LIN {X 0,Y 411.995,Z 195.318,A -85,B 0,C 180,E1 -10499.219,E2 -10499.219} C_VEL
LIN {X 0,Y 411.545,Z 202.189,A -85,B 0,C 180,E1 -10502.624,E2 -10502.624} C_VEL
LIN {X 0,Y 411.166,Z 208.718,A -85,B 0,C 180,E1 -10505.781,E2 -10505.781} C_VEL
LIN {X 0,Y 410.854,Z 215.36,A -85,B 0,C 180,E1 -10508.947,E2 -10508.947} C_VEL
LIN {X 0,Y 410.565,Z 222.705,A -85,B 0,C 180,E1 -10512.421,E2 -10512.421} C_VEL
LIN {X 0,Y 412.997,Z 235.986,A -85,B 0,C 180,E1 -10512.93,E2 -10512.93} C_VEL
LIN {X 0,Y 414.87,Z 248.726,A -85,B 0,C 180,E1 -10513.605,E2 -10513.605} C_VEL
LIN {X 0,Y 414.456,Z 259.342,A -85,B 0,C 180,E1 -10514.257,E2 -10514.257} C_VEL
LIN {X 0,Y 413.6,Z 271.793,A -85,B 0,C 180,E1 -10515.233,E2 -10515.233} C_VEL
LIN {X 0,Y 412.816,Z 282.706,A -85,B 0,C 180,E1 -10516.337,E2 -10516.337} C_VEL
LIN {X 0,Y 412.22,Z 291.609,A -85,B 0,C 180,E1 -10517.445,E2 -10517.445} C_VEL
LIN {X 0,Y 411.418,Z 301.28,A -85,B 0,C 180,E1 -10518.92,E2 -10518.92} C_VEL
LIN {X 0,Y 410.866,Z 308.982,A -85,B 0,C 180,E1 -10520.399,E2 -10520.399} C_VEL
LIN {X 0,Y 410.366,Z 316.083,A -85,B 0,C 180,E1 -10522.125,E2 -10522.125} C_VEL
LIN {X 0,Y 410.126,Z 320.996,A -85,B 0,C 180,E1 -10523.669,E2 -10523.669} C_VEL
LIN {X 0,Y 410.061,Z 324.424,A -85,B 0,C 180,E1 -10525.084,E2 -10525.084} C_VEL
LIN {X 0,Y 409.943,Z 326.285,A -85,B 0,C 180,E1 -10526.068,E2 -10526.068} C_VEL
LIN {X 0,Y 409.963,Z 328.683,A -85,B 0,C 180,E1 -10528.035,E2 -10528.035} C_VEL
LIN {X 0,Y 409.919,Z 329.291,A -85,B 0,C 180,E1 -10529.017,E2 -10529.017} C_VEL
LIN {X 0,Y 409.888,Z 329.507,A -85,B 0,C 180,E1 -10530,E2 -10530} C_VEL
LIN {X 0,Y 409.918,Z 329.292,A -85,B 0,C 180,E1 -10530.982,E2 -10530.982} C_VEL
LIN {X 0,Y 409.963,Z 328.685,A -85,B 0,C 180,E1 -10531.965,E2 -10531.965} C_VEL
LIN {X 0,Y 409.943,Z 326.29,A -85,B 0,C 180,E1 -10533.932,E2 -10533.932} C_VEL
LIN {X 0,Y 410.063,Z 323.353,A -85,B 0,C 180,E1 -10535.409,E2 -10535.409} C_VEL
LIN {X 0,Y 410.198,Z 319.375,A -85,B 0,C 180,E1 -10536.888,E2 -10536.888} C_VEL
LIN {X 0,Y 410.575,Z 313.264,A -85,B 0,C 180,E1 -10538.614,E2 -10538.614} C_VEL
LIN {X 0,Y 411.025,Z 306.584,A -85,B 0,C 180,E1 -10540.094,E2 -10540.094} C_VEL
LIN {X 0,Y 411.628,Z 298.299,A -85,B 0,C 180,E1 -10541.573,E2 -10541.573} C_VEL
LIN {X 0,Y 412.349,Z 289.811,A -85,B 0,C 180,E1 -10542.801,E2 -10542.801} C_VEL
LIN {X 0,Y 413.082,Z 279.223,A -85,B 0,C 180,E1 -10544.041,E2 -10544.041} C_VEL
LIN {X 0,Y 413.869,Z 267.514,A -85,B 0,C 180,E1 -10545.134,E2 -10545.134} C_VEL
LIN {X 0,Y 414.693,Z 255.785,A -85,B 0,C 180,E1 -10545.977,E2 -10545.977} C_VEL
LIN {X 0,Y 414.853,Z 248.666,A -85,B 0,C 180,E1 -10546.398,E2 -10546.398} C_VEL
LIN {X 0,Y 412.873,Z 235.293,A -85,B 0,C 180,E1 -10547.101,E2 -10547.101} C_VEL
LIN {X 0,Y 410.566,Z 222.705,A -85,B 0,C 180,E1 -10547.578,E2 -10547.578} C_VEL
LIN {X 0,Y 410.856,Z 215.362,A -85,B 0,C 180,E1 -10551.052,E2 -10551.052} C_VEL
LIN {X 0,Y 411.17,Z 208.721,A -85,B 0,C 180,E1 -10554.219,E2 -10554.219} C_VEL
LIN {X 0,Y 411.553,Z 202.008,A -85,B 0,C 180,E1 -10557.456,E2 -10557.456} C_VEL
LIN {X 0,Y 412.003,Z 195.293,A -85,B 0,C 180,E1 -10560.78,E2 -10560.78} C_VEL
LIN {X 0,Y 412.452,Z 188.615,A -85,B 0,C 180,E1 -10564.215,E2 -10564.215} C_VEL
LIN {X 0,Y 412.517,Z 185.292,A -85,B 0,C 180,E1 -10565.999,E2 -10565.999} C_VEL
LIN {X 0,Y 412.084,Z 181.164,A -85,B 0,C 180,E1 -10568.324,E2 -10568.324} C_VEL
LIN {X 0,Y 411.209,Z 176.266,A -85,B 0,C 180,E1 -10571.316,E2 -10571.316} C_VEL
LIN {X 0,Y 411.175,Z 176.269,A -85,B 0,C 180,E1 -10574.49,E2 -10574.49} C_VEL
LIN {X 0,Y 411.175,Z 176.267,A -85,B 0,C 180,E1 -10578.194,E2 -10578.194} C_VEL
LIN {X 0,Y 411.201,Z 176.264,A -85,B 0,C 180,E1 -10580.774,E2 -10580.774} C_VEL
LIN {X 0,Y 411.193,Z 176.267,A -85,B 0,C 180,E1 -10584.471,E2 -10584.471} C_VEL
LIN {X 0,Y 411.205,Z 176.263,A -85,B 0,C 180,E1 -10586.873,E2 -10586.873} C_VEL
LIN {X 0,Y 411.231,Z 176.26,A -85,B 0,C 180,E1 -10590.644,E2 -10590.644} C_VEL
LIN {X 0,Y 411.235,Z 176.26,A -85,B 0,C 180,E1 -10593.619,E2 -10593.619} C_VEL
LIN {X 0,Y 411.193,Z 176.262,A -85,B 0,C 180,E1 -10596.852,E2 -10596.852} C_VEL
LIN {X 0,Y 411.213,Z 176.263,A -85,B 0,C 180,E1 -10600.05,E2 -10600.05} C_VEL
LIN {X 0,Y 411.261,Z 176.257,A -85,B 0,C 180,E1 -10603.131,E2 -10603.131} C_VEL
LIN {X 0,Y 411.303,Z 176.251,A -85,B 0,C 180,E1 -10606.896,E2 -10606.896} C_VEL
LIN {X 0,Y 411.285,Z 176.251,A -85,B 0,C 180,E1 -10610.161,E2 -10610.161} C_VEL
LIN {X 0,Y 411.389,Z 176.244,A -85,B 0,C 180,E1 -10613.132,E2 -10613.132} C_VEL
LIN {X 0,Y 411.298,Z 176.254,A -85,B 0,C 180,E1 -10615.099,E2 -10615.099} C_VEL
LIN {X 0,Y 411.509,Z 176.224,A -85,B 0,C 180,E1 -10618.043,E2 -10618.043} C_VEL
LIN {X 0,Y 411.64,Z 176.208,A -85,B 0,C 180,E1 -10620,E2 -10620} C_VEL
LIN {X 0,Y 411.453,Z 176.235,A -85,B 0,C 180,E1 -10622.937,E2 -10622.937} C_VEL
LIN {X 0,Y 411.388,Z 176.239,A -85,B 0,C 180,E1 -10626.574,E2 -10626.574} C_VEL
LIN {X 0,Y 411.286,Z 176.251,A -85,B 0,C 180,E1 -10629.839,E2 -10629.839} C_VEL
LIN {X 0,Y 411.303,Z 176.249,A -85,B 0,C 180,E1 -10633.104,E2 -10633.104} C_VEL
LIN {X 0,Y 411.255,Z 176.256,A -85,B 0,C 180,E1 -10636.889,E2 -10636.889} C_VEL
LIN {X 0,Y 411.229,Z 176.263,A -85,B 0,C 180,E1 -10639.987,E2 -10639.987} C_VEL
LIN {X 0,Y 411.2,Z 176.262,A -85,B 0,C 180,E1 -10643.148,E2 -10643.148} C_VEL
LIN {X 0,Y 411.235,Z 176.258,A -85,B 0,C 180,E1 -10646.381,E2 -10646.381} C_VEL
LIN {X 0,Y 411.199,Z 176.266,A -85,B 0,C 180,E1 -10649.713,E2 -10649.713} C_VEL
LIN {X 0,Y 411.205,Z 176.265,A -85,B 0,C 180,E1 -10653.156,E2 -10653.156} C_VEL
LIN {X 0,Y 411.187,Z 176.264,A -85,B 0,C 180,E1 -10656.552,E2 -10656.552} C_VEL
LIN {X 0,Y 411.198,Z 176.263,A -85,B 0,C 180,E1 -10659.726,E2 -10659.726} C_VEL
LIN {X 0,Y 411.172,Z 176.269,A -85,B 0,C 180,E1 -10663.134,E2 -10663.134} C_VEL
LIN {X 0,Y 411.168,Z 176.266,A -85,B 0,C 180,E1 -10665.881,E2 -10665.881} C_VEL
LIN {X 0,Y 411.163,Z 176.271,A -85,B 0,C 180,E1 -10668.772,E2 -10668.772} C_VEL
LIN {X 0,Y 411.185,Z 176.265,A -85,B 0,C 180,E1 -10672.026,E2 -10672.026} C_VEL
LIN {X 0,Y 411.148,Z 176.274,A -85,B 0,C 180,E1 -10673.456,E2 -10673.456} C_VEL
LIN {X 0,Y 411.077,Z 176.794,A -85,B 0,C 180,E1 -10674.46,E2 -10674.46} C_VEL
LIN {X 0,Y 411.058,Z 179.773,A -85,B 0,C 180,E1 -10676.906,E2 -10676.906} C_VEL
LIN {X 0,Y 410.962,Z 182.568,A -85,B 0,C 180,E1 -10679.134,E2 -10679.134} C_VEL
LIN {X 0,Y 410.777,Z 186.857,A -85,B 0,C 180,E1 -10682.488,E2 -10682.488} C_VEL
LIN {X 0,Y 410.625,Z 191.146,A -85,B 0,C 180,E1 -10685.747,E2 -10685.747} C_VEL
LIN {X 0,Y 410.456,Z 195.501,A -85,B 0,C 180,E1 -10688.927,E2 -10688.927} C_VEL
LIN {X 0,Y 410.314,Z 199.943,A -85,B 0,C 180,E1 -10692.043,E2 -10692.043} C_VEL
LIN {X 0,Y 410.322,Z 200.711,A -85,B 0,C 180,E1 -10692.492,E2 -10692.492} C_VEL
LIN {X 0,Y 413.415,Z 213.717,A -85,B 0,C 180,E1 -10693.057,E2 -10693.057} C_VEL
LIN {X 0,Y 415.382,Z 224.05,A -85,B 0,C 180,E1 -10693.632,E2 -10693.632} C_VEL
LIN {X 0,Y 414.694,Z 236.478,A -85,B 0,C 180,E1 -10694.393,E2 -10694.393} C_VEL
LIN {X 0,Y 414.053,Z 247.239,A -85,B 0,C 180,E1 -10695.25,E2 -10695.25} C_VEL
LIN {X 0,Y 413.373,Z 258.203,A -85,B 0,C 180,E1 -10696.356,E2 -10696.356} C_VEL
LIN {X 0,Y 412.634,Z 267.106,A -85,B 0,C 180,E1 -10697.458,E2 -10697.458} C_VEL
LIN {X 0,Y 412.026,Z 275.27,A -85,B 0,C 180,E1 -10698.688,E2 -10698.688} C_VEL
LIN {X 0,Y 411.384,Z 283.268,A -85,B 0,C 180,E1 -10700.164,E2 -10700.164} C_VEL
LIN {X 0,Y 410.825,Z 289.69,A -85,B 0,C 180,E1 -10701.639,E2 -10701.639} C_VEL
LIN {X 0,Y 410.499,Z 295.069,A -85,B 0,C 180,E1 -10703.217,E2 -10703.217} C_VEL
LIN {X 0,Y 410.287,Z 298.734,A -85,B 0,C 180,E1 -10704.594,E2 -10704.594} C_VEL
LIN {X 0,Y 410.085,Z 301.656,A -85,B 0,C 180,E1 -10706.069,E2 -10706.069} C_VEL
LIN {X 0,Y 410.088,Z 303.054,A -85,B 0,C 180,E1 -10707.053,E2 -10707.053} C_VEL
LIN {X 0,Y 409.94,Z 304.665,A -85,B 0,C 180,E1 -10709.018,E2 -10709.018} C_VEL
LIN {X 0,Y 409.928,Z 304.899,A -85,B 0,C 180,E1 -10710,E2 -10710} C_VEL
LIN {X 0,Y 409.94,Z 304.711,A -85,B 0,C 180,E1 -10710.983,E2 -10710.983} C_VEL
LIN {X 0,Y 410.088,Z 303.159,A -85,B 0,C 180,E1 -10712.947,E2 -10712.947} C_VEL
LIN {X 0,Y 410.081,Z 301.806,A -85,B 0,C 180,E1 -10713.931,E2 -10713.931} C_VEL
LIN {X 0,Y 410.281,Z 298.941,A -85,B 0,C 180,E1 -10715.406,E2 -10715.406} C_VEL
LIN {X 0,Y 410.502,Z 295.058,A -85,B 0,C 180,E1 -10716.883,E2 -10716.883} C_VEL
LIN {X 0,Y 410.803,Z 290.048,A -85,B 0,C 180,E1 -10718.362,E2 -10718.362} C_VEL
LIN {X 0,Y 411,Z 287.371,A -85,B 0,C 180,E1 -10719.027,E2 -10719.027} C_VEL
LIN {X 0,Y 410.607,Z 284.395,A -85,B 0,C 180,E1 -10719.738,E2 -10719.738} C_VEL
LIN {X 0,Y 408.245,Z 279.193,A -85,B 0,C 180,E1 -10720.875,E2 -10720.875} C_VEL
LIN {X 0,Y 405.913,Z 273.342,A -85,B 0,C 180,E1 -10721.956,E2 -10721.956} C_VEL
LIN {X 0,Y 405.565,Z 269.345,A -85,B 0,C 180,E1 -10722.571,E2 -10722.571} C_VEL
LIN {X 0,Y 406.415,Z 259.228,A -85,B 0,C 180,E1 -10723.883,E2 -10723.883} C_VEL
LIN {X 0,Y 407.141,Z 248.492,A -85,B 0,C 180,E1 -10725.007,E2 -10725.007} C_VEL
LIN {X 0,Y 407.865,Z 238.022,A -85,B 0,C 180,E1 -10725.876,E2 -10725.876} C_VEL
LIN {X 0,Y 408.549,Z 225.844,A -85,B 0,C 180,E1 -10726.658,E2 -10726.658} C_VEL
LIN {X 0,Y 406.426,Z 214.142,A -85,B 0,C 180,E1 -10727.333,E2 -10727.333} C_VEL
LIN {X 0,Y 403.243,Z 200.765,A -85,B 0,C 180,E1 -10727.947,E2 -10727.947} C_VEL
LIN {X 0,Y 403.339,Z 197.299,A -85,B 0,C 180,E1 -10730.395,E2 -10730.395} C_VEL
LIN {X 0,Y 403.506,Z 192.933,A -85,B 0,C 180,E1 -10733.616,E2 -10733.616} C_VEL
LIN {X 0,Y 403.701,Z 188.588,A -85,B 0,C 180,E1 -10736.913,E2 -10736.913} C_VEL
LIN {X 0,Y 403.872,Z 184.3,A -85,B 0,C 180,E1 -10740.308,E2 -10740.308} C_VEL
LIN {X 0,Y 404.054,Z 179.961,A -85,B 0,C 180,E1 -10743.821,E2 -10743.821} C_VEL
LIN {X 0,Y 404.059,Z 177.157,A -85,B 0,C 180,E1 -10746.255,E2 -10746.255} C_VEL
LIN {X 0,Y 404.133,Z 177.143,A -85,B 0,C 180,E1 -10748.76,E2 -10748.76} C_VEL
LIN {X 0,Y 404.11,Z 177.148,A -85,B 0,C 180,E1 -10751.597,E2 -10751.597} C_VEL
LIN {X 0,Y 404.145,Z 177.142,A -85,B 0,C 180,E1 -10754.522,E2 -10754.522} C_VEL
LIN {X 0,Y 404.138,Z 177.145,A -85,B 0,C 180,E1 -10757.295,E2 -10757.295} C_VEL
LIN {X 0,Y 404.136,Z 177.141,A -85,B 0,C 180,E1 -10759.951,E2 -10759.951} C_VEL
LIN {X 0,Y 404.133,Z 177.145,A -85,B 0,C 180,E1 -10763.126,E2 -10763.126} C_VEL
LIN {X 0,Y 404.138,Z 177.144,A -85,B 0,C 180,E1 -10766.187,E2 -10766.187} C_VEL
LIN {X 0,Y 404.147,Z 177.141,A -85,B 0,C 180,E1 -10769.715,E2 -10769.715} C_VEL
LIN {X 0,Y 404.196,Z 177.134,A -85,B 0,C 180,E1 -10773.123,E2 -10773.123} C_VEL
LIN {X 0,Y 404.178,Z 177.136,A -85,B 0,C 180,E1 -10775.334,E2 -10775.334} C_VEL
LIN {X 0,Y 404.14,Z 177.143,A -85,B 0,C 180,E1 -10778.581,E2 -10778.581} C_VEL
LIN {X 0,Y 404.21,Z 177.137,A -85,B 0,C 180,E1 -10781.762,E2 -10781.762} C_VEL
LIN {X 0,Y 404.207,Z 177.133,A -85,B 0,C 180,E1 -10784.882,E2 -10784.882} C_VEL
LIN {X 0,Y 404.256,Z 177.13,A -85,B 0,C 180,E1 -10787.958,E2 -10787.958} C_VEL
LIN {X 0,Y 404.265,Z 177.126,A -85,B 0,C 180,E1 -10790.998,E2 -10790.998} C_VEL
LIN {X 0,Y 404.38,Z 177.113,A -85,B 0,C 180,E1 -10794.014,E2 -10794.014} C_VEL
LIN {X 0,Y 404.48,Z 177.1,A -85,B 0,C 180,E1 -10798.008,E2 -10798.008} C_VEL
LIN {X 0,Y 404.613,Z 177.083,A -85,B 0,C 180,E1 -10800,E2 -10800} C_VEL
LIN {X 0,Y 404.414,Z 177.111,A -85,B 0,C 180,E1 -10802.988,E2 -10802.988} C_VEL
LIN {X 0,Y 404.381,Z 177.111,A -85,B 0,C 180,E1 -10805.986,E2 -10805.986} C_VEL
LIN {X 0,Y 404.265,Z 177.129,A -85,B 0,C 180,E1 -10809.002,E2 -10809.002} C_VEL
LIN {X 0,Y 404.269,Z 177.126,A -85,B 0,C 180,E1 -10812.041,E2 -10812.041} C_VEL
LIN {X 0,Y 404.209,Z 177.134,A -85,B 0,C 180,E1 -10815.118,E2 -10815.118} C_VEL
LIN {X 0,Y 404.209,Z 177.136,A -85,B 0,C 180,E1 -10818.238,E2 -10818.238} C_VEL
LIN {X 0,Y 404.139,Z 177.141,A -85,B 0,C 180,E1 -10821.419,E2 -10821.419} C_VEL
LIN {X 0,Y 404.175,Z 177.138,A -85,B 0,C 180,E1 -10824.666,E2 -10824.666} C_VEL
LIN {X 0,Y 404.196,Z 177.139,A -85,B 0,C 180,E1 -10828,E2 -10828} C_VEL
LIN {X 0,Y 404.14,Z 177.145,A -85,B 0,C 180,E1 -10831.558,E2 -10831.558} C_VEL
LIN {X 0,Y 404.183,Z 177.137,A -85,B 0,C 180,E1 -10835.016,E2 -10835.016} C_VEL
LIN {X 0,Y 404.141,Z 177.141,A -85,B 0,C 180,E1 -10838.759,E2 -10838.759} C_VEL
LIN {X 0,Y 404.123,Z 177.147,A -85,B 0,C 180,E1 -10841.599,E2 -10841.599} C_VEL
LIN {X 0,Y 404.146,Z 177.144,A -85,B 0,C 180,E1 -10844.522,E2 -10844.522} C_VEL
LIN {X 0,Y 404.138,Z 177.141,A -85,B 0,C 180,E1 -10847.296,E2 -10847.296} C_VEL
LIN {X 0,Y 404.175,Z 177.178,A -85,B 0,C 180,E1 -10848.476,E2 -10848.476} C_VEL
LIN {X 0,Y 405.012,Z 181.869,A -85,B 0,C 180,E1 -10851.34,E2 -10851.34} C_VEL
LIN {X 0,Y 405.506,Z 186.296,A -85,B 0,C 180,E1 -10853.895,E2 -10853.895} C_VEL
LIN {X 0,Y 405.333,Z 190.794,A -85,B 0,C 180,E1 -10856.332,E2 -10856.332} C_VEL
LIN {X 0,Y 404.908,Z 197.401,A -85,B 0,C 180,E1 -10859.778,E2 -10859.778} C_VEL
LIN {X 0,Y 404.428,Z 204.105,A -85,B 0,C 180,E1 -10863.139,E2 -10863.139} C_VEL
LIN {X 0,Y 404.035,Z 210.759,A -85,B 0,C 180,E1 -10866.417,E2 -10866.417} C_VEL
LIN {X 0,Y 403.676,Z 218.305,A -85,B 0,C 180,E1 -10870.076,E2 -10870.076} C_VEL
LIN {X 0,Y 403.509,Z 222.624,A -85,B 0,C 180,E1 -10872.107,E2 -10872.107} C_VEL
LIN {X 0,Y 405.941,Z 235.864,A -85,B 0,C 180,E1 -10872.628,E2 -10872.628} C_VEL
LIN {X 0,Y 407.949,Z 249.164,A -85,B 0,C 180,E1 -10873.356,E2 -10873.356} C_VEL
LIN {X 0,Y 407.826,Z 255.801,A -85,B 0,C 180,E1 -10873.761,E2 -10873.761} C_VEL
LIN {X 0,Y 407.042,Z 267.3,A -85,B 0,C 180,E1 -10874.605,E2 -10874.605} C_VEL
LIN {X 0,Y 406.111,Z 279.11,A -85,B 0,C 180,E1 -10875.724,E2 -10875.724} C_VEL
LIN {X 0,Y 405.412,Z 289.597,A -85,B 0,C 180,E1 -10876.976,E2 -10876.976} C_VEL
LIN {X 0,Y 404.65,Z 298.084,A -85,B 0,C 180,E1 -10878.224,E2 -10878.224} C_VEL
LIN {X 0,Y 404.022,Z 306.369,A -85,B 0,C 180,E1 -10879.729,E2 -10879.729} C_VEL
LIN {X 0,Y 403.535,Z 313.049,A -85,B 0,C 180,E1 -10881.234,E2 -10881.234} C_VEL
LIN {X 0,Y 403.186,Z 319.164,A -85,B 0,C 180,E1 -10882.991,E2 -10882.991} C_VEL
LIN {X 0,Y 402.968,Z 323.137,A -85,B 0,C 180,E1 -10884.495,E2 -10884.495} C_VEL
LIN {X 0,Y 402.865,Z 326.073,A -85,B 0,C 180,E1 -10885.998,E2 -10885.998} C_VEL
LIN {X 0,Y 402.861,Z 328.47,A -85,B 0,C 180,E1 -10888,E2 -10888} C_VEL
LIN {X 0,Y 402.847,Z 329.079,A -85,B 0,C 180,E1 -10889,E2 -10889} C_VEL
LIN {X 0,Y 402.814,Z 329.295,A -85,B 0,C 180,E1 -10890,E2 -10890} C_VEL
LIN {X 0,Y 402.847,Z 329.08,A -85,B 0,C 180,E1 -10890.999,E2 -10890.999} C_VEL
LIN {X 0,Y 402.861,Z 328.472,A -85,B 0,C 180,E1 -10891.999,E2 -10891.999} C_VEL
LIN {X 0,Y 402.865,Z 326.077,A -85,B 0,C 180,E1 -10894.001,E2 -10894.001} C_VEL
LIN {X 0,Y 402.967,Z 323.139,A -85,B 0,C 180,E1 -10895.504,E2 -10895.504} C_VEL
LIN {X 0,Y 403.118,Z 319.161,A -85,B 0,C 180,E1 -10897.01,E2 -10897.01} C_VEL
LIN {X 0,Y 403.534,Z 313.049,A -85,B 0,C 180,E1 -10898.765,E2 -10898.765} C_VEL
LIN {X 0,Y 404.022,Z 306.37,A -85,B 0,C 180,E1 -10900.27,E2 -10900.27} C_VEL
LIN {X 0,Y 404.648,Z 298.084,A -85,B 0,C 180,E1 -10901.775,E2 -10901.775} C_VEL
LIN {X 0,Y 405.391,Z 289.595,A -85,B 0,C 180,E1 -10903.024,E2 -10903.024} C_VEL
LIN {X 0,Y 406.149,Z 278.895,A -85,B 0,C 180,E1 -10904.298,E2 -10904.298} C_VEL
LIN {X 0,Y 407.002,Z 267.297,A -85,B 0,C 180,E1 -10905.396,E2 -10905.396} C_VEL
LIN {X 0,Y 407.834,Z 255.791,A -85,B 0,C 180,E1 -10906.238,E2 -10906.238} C_VEL
LIN {X 0,Y 407.943,Z 249.145,A -85,B 0,C 180,E1 -10906.644,E2 -10906.644} C_VEL
LIN {X 0,Y 405.94,Z 235.76,A -85,B 0,C 180,E1 -10907.375,E2 -10907.375} C_VEL
LIN {X 0,Y 403.49,Z 222.465,A -85,B 0,C 180,E1 -10907.91,E2 -10907.91} C_VEL
LIN {X 0,Y 403.811,Z 215.177,A -85,B 0,C 180,E1 -10911.437,E2 -10911.437} C_VEL
LIN {X 0,Y 404.165,Z 208.55,A -85,B 0,C 180,E1 -10914.666,E2 -10914.666} C_VEL
LIN {X 0,Y 404.571,Z 201.851,A -85,B 0,C 180,E1 -10917.971,E2 -10917.971} C_VEL
LIN {X 0,Y 405.037,Z 195.146,A -85,B 0,C 180,E1 -10921.368,E2 -10921.368} C_VEL
LIN {X 0,Y 405.503,Z 188.486,A -85,B 0,C 180,E1 -10924.885,E2 -10924.885} C_VEL
LIN {X 0,Y 405.35,Z 184.521,A -85,B 0,C 180,E1 -10927.103,E2 -10927.103} C_VEL
LIN {X 0,Y 404.593,Z 179.379,A -85,B 0,C 180,E1 -10930.155,E2 -10930.155} C_VEL
LIN {X 0,Y 404.157,Z 177.145,A -85,B 0,C 180,E1 -10931.605,E2 -10931.605} C_VEL
LIN {X 0,Y 404.144,Z 177.145,A -85,B 0,C 180,E1 -10934.522,E2 -10934.522} C_VEL
LIN {X 0,Y 404.135,Z 177.143,A -85,B 0,C 180,E1 -10937.295,E2 -10937.295} C_VEL
LIN {X 0,Y 404.133,Z 177.143,A -85,B 0,C 180,E1 -10939.951,E2 -10939.951} C_VEL
LIN {X 0,Y 404.13,Z 177.143,A -85,B 0,C 180,E1 -10943.126,E2 -10943.126} C_VEL
LIN {X 0,Y 404.143,Z 177.146,A -85,B 0,C 180,E1 -10946.187,E2 -10946.187} C_VEL
LIN {X 0,Y 404.144,Z 177.144,A -85,B 0,C 180,E1 -10949.715,E2 -10949.715} C_VEL
LIN {X 0,Y 404.193,Z 177.135,A -85,B 0,C 180,E1 -10953.123,E2 -10953.123} C_VEL
LIN {X 0,Y 404.172,Z 177.138,A -85,B 0,C 180,E1 -10955.334,E2 -10955.334} C_VEL
LIN {X 0,Y 404.136,Z 177.141,A -85,B 0,C 180,E1 -10958.58,E2 -10958.58} C_VEL
LIN {X 0,Y 404.208,Z 177.137,A -85,B 0,C 180,E1 -10961.762,E2 -10961.762} C_VEL
LIN {X 0,Y 404.204,Z 177.135,A -85,B 0,C 180,E1 -10964.882,E2 -10964.882} C_VEL
LIN {X 0,Y 404.253,Z 177.128,A -85,B 0,C 180,E1 -10967.958,E2 -10967.958} C_VEL
LIN {X 0,Y 404.261,Z 177.129,A -85,B 0,C 180,E1 -10970.998,E2 -10970.998} C_VEL
LIN {X 0,Y 404.377,Z 177.111,A -85,B 0,C 180,E1 -10974.014,E2 -10974.014} C_VEL
LIN {X 0,Y 404.478,Z 177.099,A -85,B 0,C 180,E1 -10978.009,E2 -10978.009} C_VEL
LIN {X 0,Y 404.61,Z 177.083,A -85,B 0,C 180,E1 -10980,E2 -10980} C_VEL
LIN {X 0,Y 404.411,Z 177.112,A -85,B 0,C 180,E1 -10982.989,E2 -10982.989} C_VEL
LIN {X 0,Y 404.34,Z 177.116,A -85,B 0,C 180,E1 -10986.571,E2 -10986.571} C_VEL
LIN {X 0,Y 404.261,Z 177.127,A -85,B 0,C 180,E1 -10989.002,E2 -10989.002} C_VEL
LIN {X 0,Y 404.253,Z 177.13,A -85,B 0,C 180,E1 -10992.042,E2 -10992.042} C_VEL
LIN {X 0,Y 404.204,Z 177.134,A -85,B 0,C 180,E1 -10995.118,E2 -10995.118} C_VEL
LIN {X 0,Y 404.208,Z 177.138,A -85,B 0,C 180,E1 -10998.238,E2 -10998.238} C_VEL
LIN {X 0,Y 404.137,Z 177.143,A -85,B 0,C 180,E1 -11001.42,E2 -11001.42} C_VEL
LIN {X 0,Y 404.175,Z 177.136,A -85,B 0,C 180,E1 -11004.666,E2 -11004.666} C_VEL
LIN {X 0,Y 404.194,Z 177.138,A -85,B 0,C 180,E1 -11008,E2 -11008} C_VEL
LIN {X 0,Y 404.138,Z 177.146,A -85,B 0,C 180,E1 -11011.558,E2 -11011.558} C_VEL
LIN {X 0,Y 404.181,Z 177.139,A -85,B 0,C 180,E1 -11015.017,E2 -11015.017} C_VEL
LIN {X 0,Y 404.143,Z 177.143,A -85,B 0,C 180,E1 -11018.758,E2 -11018.758} C_VEL
LIN {X 0,Y 404.12,Z 177.145,A -85,B 0,C 180,E1 -11021.6,E2 -11021.6} C_VEL
LIN {X 0,Y 404.145,Z 177.143,A -85,B 0,C 180,E1 -11024.522,E2 -11024.522} C_VEL
LIN {X 0,Y 404.136,Z 177.144,A -85,B 0,C 180,E1 -11027.296,E2 -11027.296} C_VEL
LIN {X 0,Y 404.169,Z 177.138,A -85,B 0,C 180,E1 -11029.956,E2 -11029.956} C_VEL
LIN {X 0,Y 404.107,Z 177.152,A -85,B 0,C 180,E1 -11033.131,E2 -11033.131} C_VEL
LIN {X 0,Y 404.052,Z 177.158,A -85,B 0,C 180,E1 -11033.745,E2 -11033.745} C_VEL
LIN {X 0,Y 404.029,Z 179.834,A -85,B 0,C 180,E1 -11036.177,E2 -11036.177} C_VEL
LIN {X 0,Y 403.87,Z 184.136,A -85,B 0,C 180,E1 -11039.692,E2 -11039.692} C_VEL
LIN {X 0,Y 403.706,Z 188.447,A -85,B 0,C 180,E1 -11043.088,E2 -11043.088} C_VEL
LIN {X 0,Y 403.518,Z 192.774,A -85,B 0,C 180,E1 -11046.386,E2 -11046.386} C_VEL
LIN {X 0,Y 403.356,Z 197.159,A -85,B 0,C 180,E1 -11049.606,E2 -11049.606} C_VEL
LIN {X 0,Y 403.259,Z 200.784,A -85,B 0,C 180,E1 -11052.167,E2 -11052.167} C_VEL
LIN {X 0,Y 406.508,Z 214.539,A -85,B 0,C 180,E1 -11052.786,E2 -11052.786} C_VEL
LIN {X 0,Y 408.522,Z 224.998,A -85,B 0,C 180,E1 -11053.391,E2 -11053.391} C_VEL
LIN {X 0,Y 407.871,Z 236.698,A -85,B 0,C 180,E1 -11054.125,E2 -11054.125} C_VEL
LIN {X 0,Y 407.196,Z 247.457,A -85,B 0,C 180,E1 -11054.996,E2 -11054.996} C_VEL
LIN {X 0,Y 406.59,Z 257.344,A -85,B 0,C 180,E1 -11055.996,E2 -11055.996} C_VEL
LIN {X 0,Y 405.704,Z 267.323,A -85,B 0,C 180,E1 -11057.24,E2 -11057.24} C_VEL
LIN {X 0,Y 405.057,Z 275.486,A -85,B 0,C 180,E1 -11058.491,E2 -11058.491} C_VEL
LIN {X 0,Y 404.386,Z 283.484,A -85,B 0,C 180,E1 -11059.992,E2 -11059.992} C_VEL
LIN {X 0,Y 403.789,Z 289.905,A -85,B 0,C 180,E1 -11061.493,E2 -11061.493} C_VEL
LIN {X 0,Y 403.434,Z 295.579,A -85,B 0,C 180,E1 -11063.202,E2 -11063.202} C_VEL
LIN {X 0,Y 403.12,Z 300.011,A -85,B 0,C 180,E1 -11064.999,E2 -11064.999} C_VEL
LIN {X 0,Y 402.999,Z 301.87,A -85,B 0,C 180,E1 -11066,E2 -11066} C_VEL
LIN {X 0,Y 402.992,Z 303.268,A -85,B 0,C 180,E1 -11067.001,E2 -11067.001} C_VEL
LIN {X 0,Y 402.949,Z 304.263,A -85,B 0,C 180,E1 -11068.001,E2 -11068.001} C_VEL
LIN {X 0,Y 402.853,Z 305.112,A -85,B 0,C 180,E1 -11070,E2 -11070} C_VEL
LIN {X 0,Y 402.868,Z 304.923,A -85,B 0,C 180,E1 -11071,E2 -11071} C_VEL
LIN {X 0,Y 402.949,Z 304.338,A -85,B 0,C 180,E1 -11071.999,E2 -11071.999} C_VEL
LIN {X 0,Y 402.991,Z 303.372,A -85,B 0,C 180,E1 -11072.999,E2 -11072.999} C_VEL
LIN {X 0,Y 402.996,Z 302.019,A -85,B 0,C 180,E1 -11074,E2 -11074} C_VEL
LIN {X 0,Y 403.23,Z 299.153,A -85,B 0,C 180,E1 -11075.501,E2 -11075.501} C_VEL
LIN {X 0,Y 403.453,Z 295.27,A -85,B 0,C 180,E1 -11077.004,E2 -11077.004} C_VEL
LIN {X 0,Y 403.775,Z 290.26,A -85,B 0,C 180,E1 -11078.508,E2 -11078.508} C_VEL
LIN {X 0,Y 404.337,Z 283.949,A -85,B 0,C 180,E1 -11080.01,E2 -11080.01} C_VEL
LIN {X 0,Y 405.003,Z 276.049,A -85,B 0,C 180,E1 -11081.511,E2 -11081.511} C_VEL
LIN {X 0,Y 405.565,Z 269.345,A -85,B 0,C 180,E1 -11082.571,E2 -11082.571} C_VEL
LIN {X 0,Y 405.236,Z 265.24,A -85,B 0,C 180,E1 -11083.165,E2 -11083.165} C_VEL
LIN {X 0,Y 401.965,Z 255.479,A -85,B 0,C 180,E1 -11084.494,E2 -11084.494} C_VEL
LIN {X 0,Y 400.521,Z 249.397,A -85,B 0,C 180,E1 -11085.189,E2 -11085.189} C_VEL
LIN {X 0,Y 400.425,Z 246.121,A -85,B 0,C 180,E1 -11085.504,E2 -11085.504} C_VEL
LIN {X 0,Y 401.274,Z 234.989,A -85,B 0,C 180,E1 -11086.384,E2 -11086.384} C_VEL
LIN {X 0,Y 401.717,Z 226.649,A -85,B 0,C 180,E1 -11086.915,E2 -11086.915} C_VEL
LIN {X 0,Y 399.481,Z 214.718,A -85,B 0,C 180,E1 -11087.628,E2 -11087.628} C_VEL
LIN {X 0,Y 396.308,Z 201.827,A -85,B 0,C 180,E1 -11088.23,E2 -11088.23} C_VEL
LIN {X 0,Y 396.186,Z 200.965,A -85,B 0,C 180,E1 -11088.286,E2 -11088.286} C_VEL
LIN {X 0,Y 396.277,Z 197.497,A -85,B 0,C 180,E1 -11090.775,E2 -11090.775} C_VEL
LIN {X 0,Y 396.474,Z 193.113,A -85,B 0,C 180,E1 -11094.061,E2 -11094.061} C_VEL
LIN {X 0,Y 396.686,Z 188.485,A -85,B 0,C 180,E1 -11097.644,E2 -11097.644} C_VEL
LIN {X 0,Y 396.856,Z 184.447,A -85,B 0,C 180,E1 -11100.902,E2 -11100.902} C_VEL
LIN {X 0,Y 397.03,Z 180.081,A -85,B 0,C 180,E1 -11104.503,E2 -11104.503} C_VEL
LIN {X 0,Y 397.019,Z 178.624,A -85,B 0,C 180,E1 -11105.744,E2 -11105.744} C_VEL
LIN {X 0,Y 397.073,Z 178.026,A -85,B 0,C 180,E1 -11107.205,E2 -11107.205} C_VEL
LIN {X 0,Y 397.056,Z 178.024,A -85,B 0,C 180,E1 -11110.437,E2 -11110.437} C_VEL
LIN {X 0,Y 397.099,Z 178.02,A -85,B 0,C 180,E1 -11113.649,E2 -11113.649} C_VEL
LIN {X 0,Y 397.104,Z 178.019,A -85,B 0,C 180,E1 -11116.521,E2 -11116.521} C_VEL
LIN {X 0,Y 397.092,Z 178.02,A -85,B 0,C 180,E1 -11120.42,E2 -11120.42} C_VEL
LIN {X 0,Y 397.095,Z 178.022,A -85,B 0,C 180,E1 -11123.004,E2 -11123.004} C_VEL
LIN {X 0,Y 397.099,Z 178.021,A -85,B 0,C 180,E1 -11126.287,E2 -11126.287} C_VEL
LIN {X 0,Y 397.08,Z 178.022,A -85,B 0,C 180,E1 -11129.117,E2 -11129.117} C_VEL
LIN {X 0,Y 397.196,Z 178.01,A -85,B 0,C 180,E1 -11132.61,E2 -11132.61} C_VEL
LIN {X 0,Y 397.133,Z 178.017,A -85,B 0,C 180,E1 -11135.982,E2 -11135.982} C_VEL
LIN {X 0,Y 397.14,Z 178.016,A -85,B 0,C 180,E1 -11139.705,E2 -11139.705} C_VEL
LIN {X 0,Y 397.183,Z 178.008,A -85,B 0,C 180,E1 -11142.845,E2 -11142.845} C_VEL
LIN {X 0,Y 397.23,Z 178.002,A -85,B 0,C 180,E1 -11146.703,E2 -11146.703} C_VEL
LIN {X 0,Y 397.215,Z 178.008,A -85,B 0,C 180,E1 -11149.809,E2 -11149.809} C_VEL
LIN {X 0,Y 397.294,Z 177.994,A -85,B 0,C 180,E1 -11152.887,E2 -11152.887} C_VEL
LIN {X 0,Y 397.239,Z 178.002,A -85,B 0,C 180,E1 -11154.925,E2 -11154.925} C_VEL
LIN {X 0,Y 397.449,Z 177.975,A -85,B 0,C 180,E1 -11157.973,E2 -11157.973} C_VEL
LIN {X 0,Y 397.582,Z 177.958,A -85,B 0,C 180,E1 -11160,E2 -11160} C_VEL
LIN {X 0,Y 397.373,Z 177.989,A -85,B 0,C 180,E1 -11163.041,E2 -11163.041} C_VEL
LIN {X 0,Y 397.332,Z 177.989,A -85,B 0,C 180,E1 -11166.092,E2 -11166.092} C_VEL
LIN {X 0,Y 397.236,Z 178.004,A -85,B 0,C 180,E1 -11169.162,E2 -11169.162} C_VEL
LIN {X 0,Y 397.229,Z 178.004,A -85,B 0,C 180,E1 -11172.258,E2 -11172.258} C_VEL
LIN {X 0,Y 397.181,Z 178.008,A -85,B 0,C 180,E1 -11175.392,E2 -11175.392} C_VEL
LIN {X 0,Y 397.162,Z 178.015,A -85,B 0,C 180,E1 -11178.573,E2 -11178.573} C_VEL
LIN {X 0,Y 397.097,Z 178.02,A -85,B 0,C 180,E1 -11181.819,E2 -11181.819} C_VEL
LIN {X 0,Y 397.153,Z 178.012,A -85,B 0,C 180,E1 -11185.512,E2 -11185.512} C_VEL
LIN {X 0,Y 397.123,Z 178.017,A -85,B 0,C 180,E1 -11188.544,E2 -11188.544} C_VEL
LIN {X 0,Y 397.08,Z 178.025,A -85,B 0,C 180,E1 -11192.072,E2 -11192.072} C_VEL
LIN {X 0,Y 397.118,Z 178.02,A -85,B 0,C 180,E1 -11195.503,E2 -11195.503} C_VEL
LIN {X 0,Y 397.098,Z 178.018,A -85,B 0,C 180,E1 -11198.856,E2 -11198.856} C_VEL
LIN {X 0,Y 397.069,Z 178.022,A -85,B 0,C 180,E1 -11202.267,E2 -11202.267} C_VEL
LIN {X 0,Y 397.088,Z 178.024,A -85,B 0,C 180,E1 -11205.069,E2 -11205.069} C_VEL
LIN {X 0,Y 397.122,Z 178.09,A -85,B 0,C 180,E1 -11208.197,E2 -11208.197} C_VEL
LIN {X 0,Y 397.919,Z 182.557,A -85,B 0,C 180,E1 -11210.998,E2 -11210.998} C_VEL
LIN {X 0,Y 398.376,Z 186.174,A -85,B 0,C 180,E1 -11213.143,E2 -11213.143} C_VEL
LIN {X 0,Y 398.495,Z 189.489,A -85,B 0,C 180,E1 -11215.027,E2 -11215.027} C_VEL
LIN {X 0,Y 398.106,Z 195.044,A -85,B 0,C 180,E1 -11218.021,E2 -11218.021} C_VEL
LIN {X 0,Y 397.606,Z 201.709,A -85,B 0,C 180,E1 -11221.494,E2 -11221.494} C_VEL
LIN {X 0,Y 397.18,Z 208.382,A -85,B 0,C 180,E1 -11224.87,E2 -11224.87} C_VEL
LIN {X 0,Y 396.773,Z 214.992,A -85,B 0,C 180,E1 -11228.163,E2 -11228.163} C_VEL
LIN {X 0,Y 396.466,Z 222.418,A -85,B 0,C 180,E1 -11231.778,E2 -11231.778} C_VEL
LIN {X 0,Y 398.939,Z 235.552,A -85,B 0,C 180,E1 -11232.309,E2 -11232.309} C_VEL
LIN {X 0,Y 400.87,Z 248.579,A -85,B 0,C 180,E1 -11233.032,E2 -11233.032} C_VEL
LIN {X 0,Y 401.21,Z 252.359,A -85,B 0,C 180,E1 -11233.273,E2 -11233.273} C_VEL
LIN {X 0,Y 400.411,Z 263.965,A -85,B 0,C 180,E1 -11234.083,E2 -11234.083} C_VEL
LIN {X 0,Y 399.511,Z 275.279,A -85,B 0,C 180,E1 -11235.092,E2 -11235.092} C_VEL
LIN {X 0,Y 398.701,Z 285.473,A -85,B 0,C 180,E1 -11236.233,E2 -11236.233} C_VEL
LIN {X 0,Y 397.986,Z 294.652,A -85,B 0,C 180,E1 -11237.507,E2 -11237.507} C_VEL
LIN {X 0,Y 397.17,Z 303.594,A -85,B 0,C 180,E1 -11239.034,E2 -11239.034} C_VEL
LIN {X 0,Y 396.629,Z 310.796,A -85,B 0,C 180,E1 -11240.566,E2 -11240.566} C_VEL
LIN {X 0,Y 396.259,Z 315.657,A -85,B 0,C 180,E1 -11241.843,E2 -11241.843} C_VEL
LIN {X 0,Y 395.991,Z 320.527,A -85,B 0,C 180,E1 -11243.426,E2 -11243.426} C_VEL
LIN {X 0,Y 395.886,Z 323.997,A -85,B 0,C 180,E1 -11244.907,E2 -11244.907} C_VEL
LIN {X 0,Y 395.789,Z 325.86,A -85,B 0,C 180,E1 -11245.927,E2 -11245.927} C_VEL
LIN {X 0,Y 395.76,Z 328.257,A -85,B 0,C 180,E1 -11247.964,E2 -11247.964} C_VEL
LIN {X 0,Y 395.776,Z 328.867,A -85,B 0,C 180,E1 -11248.982,E2 -11248.982} C_VEL
LIN {X 0,Y 395.744,Z 329.083,A -85,B 0,C 180,E1 -11250,E2 -11250} C_VEL
LIN {X 0,Y 395.776,Z 328.867,A -85,B 0,C 180,E1 -11251.017,E2 -11251.017} C_VEL
LIN {X 0,Y 395.76,Z 328.258,A -85,B 0,C 180,E1 -11252.035,E2 -11252.035} C_VEL
LIN {X 0,Y 395.789,Z 325.864,A -85,B 0,C 180,E1 -11254.073,E2 -11254.073} C_VEL
LIN {X 0,Y 395.871,Z 322.924,A -85,B 0,C 180,E1 -11255.603,E2 -11255.603} C_VEL
LIN {X 0,Y 396.063,Z 318.947,A -85,B 0,C 180,E1 -11257.135,E2 -11257.135} C_VEL
LIN {X 0,Y 396.48,Z 312.834,A -85,B 0,C 180,E1 -11258.922,E2 -11258.922} C_VEL
LIN {X 0,Y 397.022,Z 306.155,A -85,B 0,C 180,E1 -11260.454,E2 -11260.454} C_VEL
LIN {X 0,Y 397.68,Z 297.868,A -85,B 0,C 180,E1 -11261.984,E2 -11261.984} C_VEL
LIN {X 0,Y 398.439,Z 289.379,A -85,B 0,C 180,E1 -11263.256,E2 -11263.256} C_VEL
LIN {X 0,Y 399.17,Z 279.6,A -85,B 0,C 180,E1 -11264.451,E2 -11264.451} C_VEL
LIN {X 0,Y 400.033,Z 268.51,A -85,B 0,C 180,E1 -11265.54,E2 -11265.54} C_VEL
LIN {X 0,Y 400.913,Z 257.384,A -85,B 0,C 180,E1 -11266.401,E2 -11266.401} C_VEL
LIN {X 0,Y 401.141,Z 250.51,A -85,B 0,C 180,E1 -11266.843,E2 -11266.843} C_VEL
LIN {X 0,Y 399.161,Z 237.109,A -85,B 0,C 180,E1 -11267.612,E2 -11267.612} C_VEL
LIN {X 0,Y 396.703,Z 223.939,A -85,B 0,C 180,E1 -11268.174,E2 -11268.174} C_VEL
LIN {X 0,Y 396.458,Z 222.267,A -85,B 0,C 180,E1 -11268.239,E2 -11268.239} C_VEL
LIN {X 0,Y 396.774,Z 214.992,A -85,B 0,C 180,E1 -11271.837,E2 -11271.837} C_VEL
LIN {X 0,Y 397.18,Z 208.378,A -85,B 0,C 180,E1 -11275.13,E2 -11275.13} C_VEL
LIN {X 0,Y 397.605,Z 201.699,A -85,B 0,C 180,E1 -11278.505,E2 -11278.505} C_VEL
LIN {X 0,Y 398.105,Z 195.005,A -85,B 0,C 180,E1 -11281.979,E2 -11281.979} C_VEL
LIN {X 0,Y 398.494,Z 189.473,A -85,B 0,C 180,E1 -11284.972,E2 -11284.972} C_VEL
LIN {X 0,Y 398.295,Z 185.161,A -85,B 0,C 180,E1 -11287.436,E2 -11287.436} C_VEL
LIN {X 0,Y 397.813,Z 181.738,A -85,B 0,C 180,E1 -11289.493,E2 -11289.493} C_VEL
LIN {X 0,Y 397.095,Z 178.025,A -85,B 0,C 180,E1 -11291.9,E2 -11291.9} C_VEL
LIN {X 0,Y 397.086,Z 178.023,A -85,B 0,C 180,E1 -11295.068,E2 -11295.068} C_VEL
LIN {X 0,Y 397.064,Z 178.024,A -85,B 0,C 180,E1 -11298.021,E2 -11298.021} C_VEL
LIN {X 0,Y 397.1,Z 178.018,A -85,B 0,C 180,E1 -11301.143,E2 -11301.143} C_VEL
LIN {X 0,Y 397.116,Z 178.02,A -85,B 0,C 180,E1 -11304.497,E2 -11304.497} C_VEL
LIN {X 0,Y 397.077,Z 178.025,A -85,B 0,C 180,E1 -11307.928,E2 -11307.928} C_VEL
LIN {X 0,Y 397.12,Z 178.017,A -85,B 0,C 180,E1 -11311.456,E2 -11311.456} C_VEL
LIN {X 0,Y 397.15,Z 178.013,A -85,B 0,C 180,E1 -11314.488,E2 -11314.488} C_VEL
LIN {X 0,Y 397.093,Z 178.021,A -85,B 0,C 180,E1 -11318.181,E2 -11318.181} C_VEL
LIN {X 0,Y 397.16,Z 178.015,A -85,B 0,C 180,E1 -11321.426,E2 -11321.426} C_VEL
LIN {X 0,Y 397.177,Z 178.009,A -85,B 0,C 180,E1 -11324.608,E2 -11324.608} C_VEL
LIN {X 0,Y 397.216,Z 178.006,A -85,B 0,C 180,E1 -11327.742,E2 -11327.742} C_VEL
LIN {X 0,Y 397.231,Z 178.004,A -85,B 0,C 180,E1 -11330.838,E2 -11330.838} C_VEL
LIN {X 0,Y 397.328,Z 177.989,A -85,B 0,C 180,E1 -11333.908,E2 -11333.908} C_VEL
LIN {X 0,Y 397.446,Z 177.975,A -85,B 0,C 180,E1 -11337.973,E2 -11337.973} C_VEL
LIN {X 0,Y 397.579,Z 177.959,A -85,B 0,C 180,E1 -11340,E2 -11340} C_VEL
LIN {X 0,Y 397.37,Z 177.988,A -85,B 0,C 180,E1 -11343.042,E2 -11343.042} C_VEL
LIN {X 0,Y 397.295,Z 177.993,A -85,B 0,C 180,E1 -11346.565,E2 -11346.565} C_VEL
LIN {X 0,Y 397.231,Z 178.002,A -85,B 0,C 180,E1 -11349.162,E2 -11349.162} C_VEL
LIN {X 0,Y 397.216,Z 178.009,A -85,B 0,C 180,E1 -11352.258,E2 -11352.258} C_VEL
LIN {X 0,Y 397.177,Z 178.009,A -85,B 0,C 180,E1 -11355.392,E2 -11355.392} C_VEL
LIN {X 0,Y 397.16,Z 178.012,A -85,B 0,C 180,E1 -11358.574,E2 -11358.574} C_VEL
LIN {X 0,Y 397.095,Z 178.023,A -85,B 0,C 180,E1 -11361.819,E2 -11361.819} C_VEL
LIN {X 0,Y 397.154,Z 178.011,A -85,B 0,C 180,E1 -11365.132,E2 -11365.132} C_VEL
LIN {X 0,Y 397.16,Z 178.015,A -85,B 0,C 180,E1 -11367.776,E2 -11367.776} C_VEL
LIN {X 0,Y 397.077,Z 178.022,A -85,B 0,C 180,E1 -11370.883,E2 -11370.883} C_VEL
LIN {X 0,Y 397.123,Z 178.015,A -85,B 0,C 180,E1 -11374.494,E2 -11374.494} C_VEL
LIN {X 0,Y 397.094,Z 178.019,A -85,B 0,C 180,E1 -11378.276,E2 -11378.276} C_VEL
LIN {X 0,Y 397.086,Z 178.023,A -85,B 0,C 180,E1 -11380.909,E2 -11380.909} C_VEL
LIN {X 0,Y 397.1,Z 178.019,A -85,B 0,C 180,E1 -11383.649,E2 -11383.649} C_VEL
LIN {X 0,Y 397.102,Z 178.021,A -85,B 0,C 180,E1 -11386.521,E2 -11386.521} C_VEL
LIN {X 0,Y 397.111,Z 178.02,A -85,B 0,C 180,E1 -11390.423,E2 -11390.423} C_VEL
LIN {X 0,Y 397.074,Z 178.027,A -85,B 0,C 180,E1 -11393.003,E2 -11393.003} C_VEL
LIN {X 0,Y 397.011,Z 178.828,A -85,B 0,C 180,E1 -11394.519,E2 -11394.519} C_VEL
LIN {X 0,Y 396.927,Z 182.881,A -85,B 0,C 180,E1 -11397.915,E2 -11397.915} C_VEL
LIN {X 0,Y 396.73,Z 187.179,A -85,B 0,C 180,E1 -11401.426,E2 -11401.426} C_VEL
LIN {X 0,Y 396.541,Z 191.506,A -85,B 0,C 180,E1 -11404.827,E2 -11404.827} C_VEL
LIN {X 0,Y 396.35,Z 195.887,A -85,B 0,C 180,E1 -11408.139,E2 -11408.139} C_VEL
LIN {X 0,Y 396.277,Z 198.854,A -85,B 0,C 180,E1 -11410.308,E2 -11410.308} C_VEL
LIN {X 0,Y 396.195,Z 201.001,A -85,B 0,C 180,E1 -11411.84,E2 -11411.84} C_VEL
LIN {X 0,Y 399.406,Z 214.441,A -85,B 0,C 180,E1 -11412.455,E2 -11412.455} C_VEL
LIN {X 0,Y 401.637,Z 225.883,A -85,B 0,C 180,E1 -11413.136,E2 -11413.136} C_VEL
LIN {X 0,Y 401.044,Z 236.918,A -85,B 0,C 180,E1 -11413.848,E2 -11413.848} C_VEL
LIN {X 0,Y 400.345,Z 247.676,A -85,B 0,C 180,E1 -11414.733,E2 -11414.733} C_VEL
LIN {X 0,Y 399.615,Z 258.637,A -85,B 0,C 180,E1 -11415.876,E2 -11415.876} C_VEL
LIN {X 0,Y 398.785,Z 267.539,A -85,B 0,C 180,E1 -11417.015,E2 -11417.015} C_VEL
LIN {X 0,Y 398.097,Z 275.703,A -85,B 0,C 180,E1 -11418.287,E2 -11418.287} C_VEL
LIN {X 0,Y 397.374,Z 283.7,A -85,B 0,C 180,E1 -11419.813,E2 -11419.813} C_VEL
LIN {X 0,Y 396.75,Z 290.121,A -85,B 0,C 180,E1 -11421.34,E2 -11421.34} C_VEL
LIN {X 0,Y 396.341,Z 296.182,A -85,B 0,C 180,E1 -11423.221,E2 -11423.221} C_VEL
LIN {X 0,Y 396.068,Z 300.224,A -85,B 0,C 180,E1 -11424.91,E2 -11424.91} C_VEL
LIN {X 0,Y 395.919,Z 302.084,A -85,B 0,C 180,E1 -11425.929,E2 -11425.929} C_VEL
LIN {X 0,Y 395.896,Z 303.482,A -85,B 0,C 180,E1 -11426.947,E2 -11426.947} C_VEL
LIN {X 0,Y 395.865,Z 304.476,A -85,B 0,C 180,E1 -11427.965,E2 -11427.965} C_VEL
LIN {X 0,Y 395.78,Z 305.324,A -85,B 0,C 180,E1 -11430,E2 -11430} C_VEL
LIN {X 0,Y 395.798,Z 305.135,A -85,B 0,C 180,E1 -11431.018,E2 -11431.018} C_VEL
LIN {X 0,Y 395.865,Z 304.55,A -85,B 0,C 180,E1 -11432.035,E2 -11432.035} C_VEL
LIN {X 0,Y 395.895,Z 303.585,A -85,B 0,C 180,E1 -11433.053,E2 -11433.053} C_VEL
LIN {X 0,Y 395.915,Z 302.231,A -85,B 0,C 180,E1 -11434.072,E2 -11434.072} C_VEL
LIN {X 0,Y 396.16,Z 299.365,A -85,B 0,C 180,E1 -11435.6,E2 -11435.6} C_VEL
LIN {X 0,Y 396.389,Z 295.482,A -85,B 0,C 180,E1 -11437.13,E2 -11437.13} C_VEL
LIN {X 0,Y 396.735,Z 290.472,A -85,B 0,C 180,E1 -11438.66,E2 -11438.66} C_VEL
LIN {X 0,Y 397.312,Z 284.161,A -85,B 0,C 180,E1 -11440.189,E2 -11440.189} C_VEL
LIN {X 0,Y 398.016,Z 276.26,A -85,B 0,C 180,E1 -11441.716,E2 -11441.716} C_VEL
LIN {X 0,Y 398.925,Z 266.43,A -85,B 0,C 180,E1 -11443.24,E2 -11443.24} C_VEL
LIN {X 0,Y 399.74,Z 256.684,A -85,B 0,C 180,E1 -11444.446,E2 -11444.446} C_VEL
LIN {X 0,Y 400.425,Z 246.121,A -85,B 0,C 180,E1 -11445.504,E2 -11445.504} C_VEL
LIN {X 0,Y 400.145,Z 241.118,A -85,B 0,C 180,E1 -11445.958,E2 -11445.958} C_VEL
LIN {X 0,Y 398.954,Z 236.156,A -85,B 0,C 180,E1 -11446.403,E2 -11446.403} C_VEL
LIN {X 0,Y 394.284,Z 222.744,A -85,B 0,C 180,E1 -11447.485,E2 -11447.485} C_VEL
LIN {X 0,Y 393.358,Z 219.167,A -85,B 0,C 180,E1 -11447.714,E2 -11447.714} C_VEL
LIN {X 0,Y 390.407,Z 206.294,A -85,B 0,C 180,E1 -11448.387,E2 -11448.387} C_VEL
LIN {X 0,Y 389.132,Z 201.18,A -85,B 0,C 180,E1 -11448.629,E2 -11448.629} C_VEL
LIN {X 0,Y 389.312,Z 196.229,A -85,B 0,C 180,E1 -11452.278,E2 -11452.278} C_VEL
LIN {X 0,Y 389.502,Z 191.834,A -85,B 0,C 180,E1 -11455.661,E2 -11455.661} C_VEL
LIN {X 0,Y 389.701,Z 187.489,A -85,B 0,C 180,E1 -11459.139,E2 -11459.139} C_VEL
LIN {X 0,Y 389.9,Z 183.127,A -85,B 0,C 180,E1 -11462.735,E2 -11462.735} C_VEL
LIN {X 0,Y 389.983,Z 179.547,A -85,B 0,C 180,E1 -11465.81,E2 -11465.81} C_VEL
LIN {X 0,Y 389.977,Z 178.911,A -85,B 0,C 180,E1 -11466.492,E2 -11466.492} C_VEL
LIN {X 0,Y 390.037,Z 178.903,A -85,B 0,C 180,E1 -11469.212,E2 -11469.212} C_VEL
LIN {X 0,Y 390.033,Z 178.898,A -85,B 0,C 180,E1 -11472.372,E2 -11472.372} C_VEL
LIN {X 0,Y 390.046,Z 178.9,A -85,B 0,C 180,E1 -11475.354,E2 -11475.354} C_VEL
LIN {X 0,Y 390.031,Z 178.898,A -85,B 0,C 180,E1 -11478.186,E2 -11478.186} C_VEL
LIN {X 0,Y 390.066,Z 178.899,A -85,B 0,C 180,E1 -11480.905,E2 -11480.905} C_VEL
LIN {X 0,Y 390.081,Z 178.897,A -85,B 0,C 180,E1 -11484.792,E2 -11484.792} C_VEL
LIN {X 0,Y 390.025,Z 178.904,A -85,B 0,C 180,E1 -11488.496,E2 -11488.496} C_VEL
LIN {X 0,Y 390.119,Z 178.891,A -85,B 0,C 180,E1 -11492.07,E2 -11492.07} C_VEL
LIN {X 0,Y 390.08,Z 178.892,A -85,B 0,C 180,E1 -11495.519,E2 -11495.519} C_VEL
LIN {X 0,Y 390.057,Z 178.895,A -85,B 0,C 180,E1 -11498.878,E2 -11498.878} C_VEL
LIN {X 0,Y 390.129,Z 178.891,A -85,B 0,C 180,E1 -11502.167,E2 -11502.167} C_VEL
LIN {X 0,Y 390.145,Z 178.887,A -85,B 0,C 180,E1 -11505.393,E2 -11505.393} C_VEL
LIN {X 0,Y 390.147,Z 178.884,A -85,B 0,C 180,E1 -11508.571,E2 -11508.571} C_VEL
LIN {X 0,Y 390.257,Z 178.871,A -85,B 0,C 180,E1 -11512.086,E2 -11512.086} C_VEL
LIN {X 0,Y 390.21,Z 178.877,A -85,B 0,C 180,E1 -11514.833,E2 -11514.833} C_VEL
LIN {X 0,Y 390.418,Z 178.851,A -85,B 0,C 180,E1 -11517.937,E2 -11517.937} C_VEL
LIN {X 0,Y 390.551,Z 178.834,A -85,B 0,C 180,E1 -11520,E2 -11520} C_VEL
LIN {X 0,Y 390.307,Z 178.869,A -85,B 0,C 180,E1 -11523.097,E2 -11523.097} C_VEL
LIN {X 0,Y 390.285,Z 178.867,A -85,B 0,C 180,E1 -11526.203,E2 -11526.203} C_VEL
LIN {X 0,Y 390.194,Z 178.879,A -85,B 0,C 180,E1 -11529.329,E2 -11529.329} C_VEL
LIN {X 0,Y 390.178,Z 178.885,A -85,B 0,C 180,E1 -11532.483,E2 -11532.483} C_VEL
LIN {X 0,Y 390.141,Z 178.885,A -85,B 0,C 180,E1 -11535.677,E2 -11535.677} C_VEL
LIN {X 0,Y 390.106,Z 178.89,A -85,B 0,C 180,E1 -11538.922,E2 -11538.922} C_VEL
LIN {X 0,Y 390.039,Z 178.903,A -85,B 0,C 180,E1 -11542.234,E2 -11542.234} C_VEL
LIN {X 0,Y 390.12,Z 178.89,A -85,B 0,C 180,E1 -11545.743,E2 -11545.743} C_VEL
LIN {X 0,Y 390.059,Z 178.895,A -85,B 0,C 180,E1 -11549.11,E2 -11549.11} C_VEL
LIN {X 0,Y 390.044,Z 178.897,A -85,B 0,C 180,E1 -11552.721,E2 -11552.721} C_VEL
LIN {X 0,Y 390.054,Z 178.9,A -85,B 0,C 180,E1 -11555.825,E2 -11555.825} C_VEL
LIN {X 0,Y 390.041,Z 178.9,A -85,B 0,C 180,E1 -11559.213,E2 -11559.213} C_VEL
LIN {X 0,Y 390.043,Z 178.897,A -85,B 0,C 180,E1 -11562.374,E2 -11562.374} C_VEL
LIN {X 0,Y 390.046,Z 178.901,A -85,B 0,C 180,E1 -11565.354,E2 -11565.354} C_VEL
LIN {X 0,Y 390.073,Z 178.987,A -85,B 0,C 180,E1 -11567.91,E2 -11567.91} C_VEL
LIN {X 0,Y 390.95,Z 183.836,A -85,B 0,C 180,E1 -11571.01,E2 -11571.01} C_VEL
LIN {X 0,Y 391.43,Z 188.257,A -85,B 0,C 180,E1 -11573.665,E2 -11573.665} C_VEL
LIN {X 0,Y 391.42,Z 191.801,A -85,B 0,C 180,E1 -11575.684,E2 -11575.684} C_VEL
LIN {X 0,Y 390.92,Z 198.221,A -85,B 0,C 180,E1 -11579.178,E2 -11579.178} C_VEL
LIN {X 0,Y 390.389,Z 204.895,A -85,B 0,C 180,E1 -11582.673,E2 -11582.673} C_VEL
LIN {X 0,Y 389.955,Z 211.504,A -85,B 0,C 180,E1 -11586.077,E2 -11586.077} C_VEL
LIN {X 0,Y 389.545,Z 219.156,A -85,B 0,C 180,E1 -11589.953,E2 -11589.953} C_VEL
LIN {X 0,Y 389.414,Z 222.211,A -85,B 0,C 180,E1 -11591.436,E2 -11591.436} C_VEL
LIN {X 0,Y 391.905,Z 235.351,A -85,B 0,C 180,E1 -11591.981,E2 -11591.981} C_VEL
LIN {X 0,Y 393.714,Z 247.567,A -85,B 0,C 180,E1 -11592.667,E2 -11592.667} C_VEL
LIN {X 0,Y 394.351,Z 252.549,A -85,B 0,C 180,E1 -11593,E2 -11593} C_VEL
LIN {X 0,Y 393.465,Z 265.341,A -85,B 0,C 180,E1 -11593.927,E2 -11593.927} C_VEL
LIN {X 0,Y 392.477,Z 276.799,A -85,B 0,C 180,E1 -11595.004,E2 -11595.004} C_VEL
LIN {X 0,Y 391.661,Z 287.328,A -85,B 0,C 180,E1 -11596.26,E2 -11596.26} C_VEL
LIN {X 0,Y 390.865,Z 296.073,A -85,B 0,C 180,E1 -11597.539,E2 -11597.539} C_VEL
LIN {X 0,Y 390.078,Z 304.706,A -85,B 0,C 180,E1 -11599.095,E2 -11599.095} C_VEL
LIN {X 0,Y 389.515,Z 311.609,A -85,B 0,C 180,E1 -11600.654,E2 -11600.654} C_VEL
LIN {X 0,Y 389.094,Z 317.142,A -85,B 0,C 180,E1 -11602.214,E2 -11602.214} C_VEL
LIN {X 0,Y 388.835,Z 321.483,A -85,B 0,C 180,E1 -11603.774,E2 -11603.774} C_VEL
LIN {X 0,Y 388.782,Z 323.784,A -85,B 0,C 180,E1 -11604.814,E2 -11604.814} C_VEL
LIN {X 0,Y 388.715,Z 325.648,A -85,B 0,C 180,E1 -11605.852,E2 -11605.852} C_VEL
LIN {X 0,Y 388.659,Z 328.044,A -85,B 0,C 180,E1 -11607.927,E2 -11607.927} C_VEL
LIN {X 0,Y 388.689,Z 328.654,A -85,B 0,C 180,E1 -11608.964,E2 -11608.964} C_VEL
LIN {X 0,Y 388.675,Z 328.871,A -85,B 0,C 180,E1 -11610,E2 -11610} C_VEL
LIN {X 0,Y 388.689,Z 328.654,A -85,B 0,C 180,E1 -11611.036,E2 -11611.036} C_VEL
LIN {X 0,Y 388.658,Z 328.045,A -85,B 0,C 180,E1 -11612.072,E2 -11612.072} C_VEL
LIN {X 0,Y 388.715,Z 325.65,A -85,B 0,C 180,E1 -11614.147,E2 -11614.147} C_VEL
LIN {X 0,Y 388.796,Z 322.375,A -85,B 0,C 180,E1 -11615.854,E2 -11615.854} C_VEL
LIN {X 0,Y 389.094,Z 317.138,A -85,B 0,C 180,E1 -11617.785,E2 -11617.785} C_VEL
LIN {X 0,Y 389.515,Z 311.605,A -85,B 0,C 180,E1 -11619.345,E2 -11619.345} C_VEL
LIN {X 0,Y 390.077,Z 304.7,A -85,B 0,C 180,E1 -11620.905,E2 -11620.905} C_VEL
LIN {X 0,Y 390.858,Z 296.065,A -85,B 0,C 180,E1 -11622.46,E2 -11622.46} C_VEL
LIN {X 0,Y 391.643,Z 287.288,A -85,B 0,C 180,E1 -11623.744,E2 -11623.744} C_VEL
LIN {X 0,Y 392.501,Z 276.786,A -85,B 0,C 180,E1 -11624.995,E2 -11624.995} C_VEL
LIN {X 0,Y 393.298,Z 266.863,A -85,B 0,C 180,E1 -11625.946,E2 -11625.946} C_VEL
LIN {X 0,Y 394.182,Z 255.748,A -85,B 0,C 180,E1 -11626.791,E2 -11626.791} C_VEL
LIN {X 0,Y 394.158,Z 250.847,A -85,B 0,C 180,E1 -11627.117,E2 -11627.117} C_VEL
LIN {X 0,Y 392.232,Z 237.559,A -85,B 0,C 180,E1 -11627.904,E2 -11627.904} C_VEL
LIN {X 0,Y 389.762,Z 224.159,A -85,B 0,C 180,E1 -11628.497,E2 -11628.497} C_VEL
LIN {X 0,Y 389.407,Z 222.055,A -85,B 0,C 180,E1 -11628.581,E2 -11628.581} C_VEL
LIN {X 0,Y 389.696,Z 215.9,A -85,B 0,C 180,E1 -11631.697,E2 -11631.697} C_VEL
LIN {X 0,Y 390.102,Z 209.308,A -85,B 0,C 180,E1 -11635.047,E2 -11635.047} C_VEL
LIN {X 0,Y 390.494,Z 203.329,A -85,B 0,C 180,E1 -11638.129,E2 -11638.129} C_VEL
LIN {X 0,Y 390.975,Z 197.091,A -85,B 0,C 180,E1 -11641.419,E2 -11641.419} C_VEL
LIN {X 0,Y 391.41,Z 191.768,A -85,B 0,C 180,E1 -11644.314,E2 -11644.314} C_VEL
LIN {X 0,Y 391.383,Z 187.13,A -85,B 0,C 180,E1 -11646.981,E2 -11646.981} C_VEL
LIN {X 0,Y 390.877,Z 183.217,A -85,B 0,C 180,E1 -11649.363,E2 -11649.363} C_VEL
LIN {X 0,Y 390.06,Z 178.9,A -85,B 0,C 180,E1 -11652.189,E2 -11652.189} C_VEL
LIN {X 0,Y 390.043,Z 178.898,A -85,B 0,C 180,E1 -11655.354,E2 -11655.354} C_VEL
LIN {X 0,Y 390.029,Z 178.901,A -85,B 0,C 180,E1 -11658.186,E2 -11658.186} C_VEL
LIN {X 0,Y 390.063,Z 178.896,A -85,B 0,C 180,E1 -11660.904,E2 -11660.904} C_VEL
LIN {X 0,Y 390.082,Z 178.894,A -85,B 0,C 180,E1 -11664.793,E2 -11664.793} C_VEL
LIN {X 0,Y 390.022,Z 178.903,A -85,B 0,C 180,E1 -11668.495,E2 -11668.495} C_VEL
LIN {X 0,Y 390.115,Z 178.893,A -85,B 0,C 180,E1 -11672.07,E2 -11672.07} C_VEL
LIN {X 0,Y 390.075,Z 178.895,A -85,B 0,C 180,E1 -11675.519,E2 -11675.519} C_VEL
LIN {X 0,Y 390.085,Z 178.896,A -85,B 0,C 180,E1 -11679.53,E2 -11679.53} C_VEL
LIN {X 0,Y 390.136,Z 178.889,A -85,B 0,C 180,E1 -11683.248,E2 -11683.248} C_VEL
LIN {X 0,Y 390.192,Z 178.879,A -85,B 0,C 180,E1 -11686.561,E2 -11686.561} C_VEL
LIN {X 0,Y 390.163,Z 178.885,A -85,B 0,C 180,E1 -11689.623,E2 -11689.623} C_VEL
LIN {X 0,Y 390.244,Z 178.874,A -85,B 0,C 180,E1 -11692.758,E2 -11692.758} C_VEL
LIN {X 0,Y 390.209,Z 178.88,A -85,B 0,C 180,E1 -11694.833,E2 -11694.833} C_VEL
LIN {X 0,Y 390.415,Z 178.851,A -85,B 0,C 180,E1 -11697.937,E2 -11697.937} C_VEL
LIN {X 0,Y 390.548,Z 178.834,A -85,B 0,C 180,E1 -11700,E2 -11700} C_VEL
LIN {X 0,Y 390.304,Z 178.867,A -85,B 0,C 180,E1 -11703.097,E2 -11703.097} C_VEL
LIN {X 0,Y 390.255,Z 178.87,A -85,B 0,C 180,E1 -11706.556,E2 -11706.556} C_VEL
LIN {X 0,Y 390.189,Z 178.878,A -85,B 0,C 180,E1 -11709.329,E2 -11709.329} C_VEL
LIN {X 0,Y 390.168,Z 178.886,A -85,B 0,C 180,E1 -11712.483,E2 -11712.483} C_VEL
LIN {X 0,Y 390.137,Z 178.887,A -85,B 0,C 180,E1 -11715.677,E2 -11715.677} C_VEL
LIN {X 0,Y 390.104,Z 178.89,A -85,B 0,C 180,E1 -11718.922,E2 -11718.922} C_VEL
LIN {X 0,Y 390.038,Z 178.9,A -85,B 0,C 180,E1 -11722.234,E2 -11722.234} C_VEL
LIN {X 0,Y 390.117,Z 178.893,A -85,B 0,C 180,E1 -11725.744,E2 -11725.744} C_VEL
LIN {X 0,Y 390.057,Z 178.897,A -85,B 0,C 180,E1 -11729.11,E2 -11729.11} C_VEL
LIN {X 0,Y 390.041,Z 178.898,A -85,B 0,C 180,E1 -11732.722,E2 -11732.722} C_VEL
LIN {X 0,Y 390.052,Z 178.898,A -85,B 0,C 180,E1 -11735.825,E2 -11735.825} C_VEL
LIN {X 0,Y 390.043,Z 178.903,A -85,B 0,C 180,E1 -11739.214,E2 -11739.214} C_VEL
LIN {X 0,Y 390.041,Z 178.897,A -85,B 0,C 180,E1 -11742.374,E2 -11742.374} C_VEL
LIN {X 0,Y 390.044,Z 178.899,A -85,B 0,C 180,E1 -11745.355,E2 -11745.355} C_VEL
LIN {X 0,Y 390.031,Z 178.9,A -85,B 0,C 180,E1 -11748.187,E2 -11748.187} C_VEL
LIN {X 0,Y 390.085,Z 178.896,A -85,B 0,C 180,E1 -11750.908,E2 -11750.908} C_VEL
LIN {X 0,Y 389.971,Z 178.912,A -85,B 0,C 180,E1 -11753.508,E2 -11753.508} C_VEL
LIN {X 0,Y 389.983,Z 180.117,A -85,B 0,C 180,E1 -11754.783,E2 -11754.783} C_VEL
LIN {X 0,Y 389.882,Z 183.772,A -85,B 0,C 180,E1 -11757.911,E2 -11757.911} C_VEL
LIN {X 0,Y 389.703,Z 187.36,A -85,B 0,C 180,E1 -11760.862,E2 -11760.862} C_VEL
LIN {X 0,Y 389.506,Z 191.689,A -85,B 0,C 180,E1 -11764.34,E2 -11764.34} C_VEL
LIN {X 0,Y 389.342,Z 196.082,A -85,B 0,C 180,E1 -11767.724,E2 -11767.724} C_VEL
LIN {X 0,Y 389.141,Z 200.574,A -85,B 0,C 180,E1 -11771.03,E2 -11771.03} C_VEL
LIN {X 0,Y 389.146,Z 201.251,A -85,B 0,C 180,E1 -11771.501,E2 -11771.501} C_VEL
LIN {X 0,Y 392.329,Z 214.343,A -85,B 0,C 180,E1 -11772.113,E2 -11772.113} C_VEL
LIN {X 0,Y 394.748,Z 226.688,A -85,B 0,C 180,E1 -11772.867,E2 -11772.867} C_VEL
LIN {X 0,Y 394.612,Z 232.688,A -85,B 0,C 180,E1 -11773.25,E2 -11773.25} C_VEL
LIN {X 0,Y 393.802,Z 243.612,A -85,B 0,C 180,E1 -11774.075,E2 -11774.075} C_VEL
LIN {X 0,Y 392.989,Z 254.643,A -85,B 0,C 180,E1 -11775.144,E2 -11775.144} C_VEL
LIN {X 0,Y 392.281,Z 264.001,A -85,B 0,C 180,E1 -11776.268,E2 -11776.268} C_VEL
LIN {X 0,Y 391.363,Z 272.844,A -85,B 0,C 180,E1 -11777.556,E2 -11777.556} C_VEL
LIN {X 0,Y 390.599,Z 281.464,A -85,B 0,C 180,E1 -11779.11,E2 -11779.11} C_VEL
LIN {X 0,Y 389.926,Z 288.337,A -85,B 0,C 180,E1 -11780.665,E2 -11780.665} C_VEL
LIN {X 0,Y 389.457,Z 293.838,A -85,B 0,C 180,E1 -11782.222,E2 -11782.222} C_VEL
LIN {X 0,Y 389.191,Z 298.153,A -85,B 0,C 180,E1 -11783.78,E2 -11783.78} C_VEL
LIN {X 0,Y 389.016,Z 300.438,A -85,B 0,C 180,E1 -11784.818,E2 -11784.818} C_VEL
LIN {X 0,Y 388.843,Z 302.298,A -85,B 0,C 180,E1 -11785.854,E2 -11785.854} C_VEL
LIN {X 0,Y 388.801,Z 303.696,A -85,B 0,C 180,E1 -11786.892,E2 -11786.892} C_VEL
LIN {X 0,Y 388.768,Z 304.69,A -85,B 0,C 180,E1 -11787.928,E2 -11787.928} C_VEL
LIN {X 0,Y 388.709,Z 305.536,A -85,B 0,C 180,E1 -11790,E2 -11790} C_VEL
LIN {X 0,Y 388.73,Z 305.347,A -85,B 0,C 180,E1 -11791.036,E2 -11791.036} C_VEL
LIN {X 0,Y 388.769,Z 304.763,A -85,B 0,C 180,E1 -11792.072,E2 -11792.072} C_VEL
LIN {X 0,Y 388.799,Z 303.797,A -85,B 0,C 180,E1 -11793.109,E2 -11793.109} C_VEL
LIN {X 0,Y 388.839,Z 302.443,A -85,B 0,C 180,E1 -11794.146,E2 -11794.146} C_VEL
LIN {X 0,Y 389.093,Z 299.577,A -85,B 0,C 180,E1 -11795.702,E2 -11795.702} C_VEL
LIN {X 0,Y 389.334,Z 295.694,A -85,B 0,C 180,E1 -11797.259,E2 -11797.259} C_VEL
LIN {X 0,Y 389.707,Z 290.684,A -85,B 0,C 180,E1 -11798.818,E2 -11798.818} C_VEL
LIN {X 0,Y 390.32,Z 284.372,A -85,B 0,C 180,E1 -11800.373,E2 -11800.373} C_VEL
LIN {X 0,Y 391.057,Z 276.471,A -85,B 0,C 180,E1 -11801.928,E2 -11801.928} C_VEL
LIN {X 0,Y 392.016,Z 266.639,A -85,B 0,C 180,E1 -11803.478,E2 -11803.478} C_VEL
LIN {X 0,Y 392.849,Z 257.224,A -85,B 0,C 180,E1 -11804.667,E2 -11804.667} C_VEL
LIN {X 0,Y 393.6,Z 246.103,A -85,B 0,C 180,E1 -11805.801,E2 -11805.801} C_VEL
LIN {X 0,Y 394.607,Z 233.853,A -85,B 0,C 180,E1 -11806.769,E2 -11806.769} C_VEL
LIN {X 0,Y 394.861,Z 227.417,A -85,B 0,C 180,E1 -11807.184,E2 -11807.184} C_VEL
LIN {X 0,Y 393.358,Z 219.167,A -85,B 0,C 180,E1 -11807.714,E2 -11807.714} C_VEL
LIN {X 0,Y 392.003,Z 215.795,A -85,B 0,C 180,E1 -11807.946,E2 -11807.946} C_VEL
LIN {X 0,Y 388.097,Z 211.026,A -85,B 0,C 180,E1 -11808.341,E2 -11808.341} C_VEL
LIN {X 0,Y 383.995,Z 206.24,A -85,B 0,C 180,E1 -11808.713,E2 -11808.713} C_VEL
LIN {X 0,Y 382.326,Z 202.822,A -85,B 0,C 180,E1 -11808.903,E2 -11808.903} C_VEL
LIN {X 0,Y 382.076,Z 201.381,A -85,B 0,C 180,E1 -11808.987,E2 -11808.987} C_VEL
LIN {X 0,Y 382.289,Z 196.422,A -85,B 0,C 180,E1 -11812.71,E2 -11812.71} C_VEL
LIN {X 0,Y 382.472,Z 192.01,A -85,B 0,C 180,E1 -11816.168,E2 -11816.168} C_VEL
LIN {X 0,Y 382.628,Z 189.103,A -85,B 0,C 180,E1 -11818.526,E2 -11818.526} C_VEL
LIN {X 0,Y 382.745,Z 186.179,A -85,B 0,C 180,E1 -11820.94,E2 -11820.94} C_VEL
LIN {X 0,Y 382.902,Z 183.286,A -85,B 0,C 180,E1 -11823.411,E2 -11823.411} C_VEL
LIN {X 0,Y 382.938,Z 180.159,A -85,B 0,C 180,E1 -11826.145,E2 -11826.145} C_VEL
LIN {X 0,Y 382.988,Z 179.777,A -85,B 0,C 180,E1 -11827.901,E2 -11827.901} C_VEL
LIN {X 0,Y 382.962,Z 179.784,A -85,B 0,C 180,E1 -11831.35,E2 -11831.35} C_VEL
LIN {X 0,Y 382.996,Z 179.775,A -85,B 0,C 180,E1 -11834.303,E2 -11834.303} C_VEL
LIN {X 0,Y 383.012,Z 179.776,A -85,B 0,C 180,E1 -11837.24,E2 -11837.24} C_VEL
LIN {X 0,Y 383.001,Z 179.775,A -85,B 0,C 180,E1 -11840.416,E2 -11840.416} C_VEL
LIN {X 0,Y 383.022,Z 179.772,A -85,B 0,C 180,E1 -11844.044,E2 -11844.044} C_VEL
LIN {X 0,Y 382.987,Z 179.776,A -85,B 0,C 180,E1 -11847.578,E2 -11847.578} C_VEL
LIN {X 0,Y 382.994,Z 179.78,A -85,B 0,C 180,E1 -11850.3,E2 -11850.3} C_VEL
LIN {X 0,Y 383.081,Z 179.767,A -85,B 0,C 180,E1 -11854.021,E2 -11854.021} C_VEL
LIN {X 0,Y 383.009,Z 179.773,A -85,B 0,C 180,E1 -11857.335,E2 -11857.335} C_VEL
LIN {X 0,Y 383.061,Z 179.767,A -85,B 0,C 180,E1 -11860.716,E2 -11860.716} C_VEL
LIN {X 0,Y 383.082,Z 179.769,A -85,B 0,C 180,E1 -11864.027,E2 -11864.027} C_VEL
LIN {X 0,Y 383.137,Z 179.759,A -85,B 0,C 180,E1 -11867.284,E2 -11867.284} C_VEL
LIN {X 0,Y 383.143,Z 179.756,A -85,B 0,C 180,E1 -11870.498,E2 -11870.498} C_VEL
LIN {X 0,Y 383.241,Z 179.748,A -85,B 0,C 180,E1 -11873.683,E2 -11873.683} C_VEL
LIN {X 0,Y 383.385,Z 179.727,A -85,B 0,C 180,E1 -11877.899,E2 -11877.899} C_VEL
LIN {X 0,Y 383.521,Z 179.71,A -85,B 0,C 180,E1 -11880,E2 -11880} C_VEL
LIN {X 0,Y 383.244,Z 179.749,A -85,B 0,C 180,E1 -11883.154,E2 -11883.154} C_VEL
LIN {X 0,Y 383.242,Z 179.745,A -85,B 0,C 180,E1 -11886.317,E2 -11886.317} C_VEL
LIN {X 0,Y 383.144,Z 179.756,A -85,B 0,C 180,E1 -11889.502,E2 -11889.502} C_VEL
LIN {X 0,Y 383.142,Z 179.762,A -85,B 0,C 180,E1 -11892.716,E2 -11892.716} C_VEL
LIN {X 0,Y 383.082,Z 179.765,A -85,B 0,C 180,E1 -11895.973,E2 -11895.973} C_VEL
LIN {X 0,Y 383.061,Z 179.766,A -85,B 0,C 180,E1 -11899.284,E2 -11899.284} C_VEL
LIN {X 0,Y 382.992,Z 179.777,A -85,B 0,C 180,E1 -11902.666,E2 -11902.666} C_VEL
LIN {X 0,Y 383.081,Z 179.769,A -85,B 0,C 180,E1 -11906.123,E2 -11906.123} C_VEL
LIN {X 0,Y 382.993,Z 179.779,A -85,B 0,C 180,E1 -11909.7,E2 -11909.7} C_VEL
LIN {X 0,Y 383.004,Z 179.776,A -85,B 0,C 180,E1 -11913.401,E2 -11913.401} C_VEL
LIN {X 0,Y 383.03,Z 179.772,A -85,B 0,C 180,E1 -11916.164,E2 -11916.164} C_VEL
LIN {X 0,Y 383,Z 179.776,A -85,B 0,C 180,E1 -11919.96,E2 -11919.96} C_VEL
LIN {X 0,Y 383.006,Z 179.774,A -85,B 0,C 180,E1 -11922.779,E2 -11922.779} C_VEL
LIN {X 0,Y 382.998,Z 179.778,A -85,B 0,C 180,E1 -11925.789,E2 -11925.789} C_VEL
LIN {X 0,Y 383.021,Z 179.857,A -85,B 0,C 180,E1 -11927.598,E2 -11927.598} C_VEL
LIN {X 0,Y 383.786,Z 183.941,A -85,B 0,C 180,E1 -11930.275,E2 -11930.275} C_VEL
LIN {X 0,Y 384.361,Z 188.127,A -85,B 0,C 180,E1 -11932.886,E2 -11932.886} C_VEL
LIN {X 0,Y 384.434,Z 192.539,A -85,B 0,C 180,E1 -11935.478,E2 -11935.478} C_VEL
LIN {X 0,Y 383.945,Z 198.068,A -85,B 0,C 180,E1 -11938.555,E2 -11938.555} C_VEL
LIN {X 0,Y 383.473,Z 203.738,A -85,B 0,C 180,E1 -11941.607,E2 -11941.607} C_VEL
LIN {X 0,Y 383.022,Z 210.228,A -85,B 0,C 180,E1 -11945.037,E2 -11945.037} C_VEL
LIN {X 0,Y 382.584,Z 217.884,A -85,B 0,C 180,E1 -11949.01,E2 -11949.01} C_VEL
LIN {X 0,Y 382.365,Z 222.004,A -85,B 0,C 180,E1 -11951.081,E2 -11951.081} C_VEL
LIN {X 0,Y 384.921,Z 235.139,A -85,B 0,C 180,E1 -11951.642,E2 -11951.642} C_VEL
LIN {X 0,Y 386.769,Z 247.626,A -85,B 0,C 180,E1 -11952.362,E2 -11952.362} C_VEL
LIN {X 0,Y 387.444,Z 254.194,A -85,B 0,C 180,E1 -11952.814,E2 -11952.814} C_VEL
LIN {X 0,Y 386.511,Z 266.67,A -85,B 0,C 180,E1 -11953.765,E2 -11953.765} C_VEL
LIN {X 0,Y 385.523,Z 277.294,A -85,B 0,C 180,E1 -11954.808,E2 -11954.808} C_VEL
LIN {X 0,Y 384.706,Z 287.326,A -85,B 0,C 180,E1 -11956.035,E2 -11956.035} C_VEL
LIN {X 0,Y 383.915,Z 295.862,A -85,B 0,C 180,E1 -11957.31,E2 -11957.31} C_VEL
LIN {X 0,Y 383.05,Z 304.493,A -85,B 0,C 180,E1 -11958.892,E2 -11958.892} C_VEL
LIN {X 0,Y 382.478,Z 311.396,A -85,B 0,C 180,E1 -11960.481,E2 -11960.481} C_VEL
LIN {X 0,Y 382.052,Z 316.929,A -85,B 0,C 180,E1 -11962.07,E2 -11962.07} C_VEL
LIN {X 0,Y 381.738,Z 321.631,A -85,B 0,C 180,E1 -11963.811,E2 -11963.811} C_VEL
LIN {X 0,Y 381.641,Z 325.435,A -85,B 0,C 180,E1 -11965.775,E2 -11965.775} C_VEL
LIN {X 0,Y 381.558,Z 327.831,A -85,B 0,C 180,E1 -11967.889,E2 -11967.889} C_VEL
LIN {X 0,Y 381.59,Z 328.441,A -85,B 0,C 180,E1 -11968.944,E2 -11968.944} C_VEL
LIN {X 0,Y 381.59,Z 328.658,A -85,B 0,C 180,E1 -11970,E2 -11970} C_VEL
LIN {X 0,Y 381.59,Z 328.441,A -85,B 0,C 180,E1 -11971.055,E2 -11971.055} C_VEL
LIN {X 0,Y 381.558,Z 327.831,A -85,B 0,C 180,E1 -11972.111,E2 -11972.111} C_VEL
LIN {X 0,Y 381.641,Z 325.437,A -85,B 0,C 180,E1 -11974.224,E2 -11974.224} C_VEL
LIN {X 0,Y 381.749,Z 321.592,A -85,B 0,C 180,E1 -11976.204,E2 -11976.204} C_VEL
LIN {X 0,Y 382.052,Z 316.923,A -85,B 0,C 180,E1 -11977.93,E2 -11977.93} C_VEL
LIN {X 0,Y 382.477,Z 311.39,A -85,B 0,C 180,E1 -11979.519,E2 -11979.519} C_VEL
LIN {X 0,Y 383.048,Z 304.484,A -85,B 0,C 180,E1 -11981.107,E2 -11981.107} C_VEL
LIN {X 0,Y 383.906,Z 295.849,A -85,B 0,C 180,E1 -11982.69,E2 -11982.69} C_VEL
LIN {X 0,Y 384.878,Z 285.567,A -85,B 0,C 180,E1 -11984.198,E2 -11984.198} C_VEL
LIN {X 0,Y 385.64,Z 276.096,A -85,B 0,C 180,E1 -11985.322,E2 -11985.322} C_VEL
LIN {X 0,Y 386.581,Z 265.104,A -85,B 0,C 180,E1 -11986.367,E2 -11986.367} C_VEL
LIN {X 0,Y 387.431,Z 254.15,A -85,B 0,C 180,E1 -11987.186,E2 -11987.186} C_VEL
LIN {X 0,Y 385.867,Z 241.046,A -85,B 0,C 180,E1 -11988.037,E2 -11988.037} C_VEL
LIN {X 0,Y 383.676,Z 228.516,A -85,B 0,C 180,E1 -11988.663,E2 -11988.663} C_VEL
LIN {X 0,Y 382.338,Z 221.844,A -85,B 0,C 180,E1 -11988.938,E2 -11988.938} C_VEL
LIN {X 0,Y 382.681,Z 215.708,A -85,B 0,C 180,E1 -11992.116,E2 -11992.116} C_VEL
LIN {X 0,Y 383.022,Z 210.233,A -85,B 0,C 180,E1 -11994.962,E2 -11994.962} C_VEL
LIN {X 0,Y 383.478,Z 203.6,A -85,B 0,C 180,E1 -11998.457,E2 -11998.457} C_VEL
LIN {X 0,Y 383.947,Z 198.044,A -85,B 0,C 180,E1 -12001.445,E2 -12001.445} C_VEL
LIN {X 0,Y 384.427,Z 192.295,A -85,B 0,C 180,E1 -12004.646,E2 -12004.646} C_VEL
LIN {X 0,Y 384.362,Z 188.096,A -85,B 0,C 180,E1 -12007.113,E2 -12007.113} C_VEL
LIN {X 0,Y 383.745,Z 183.696,A -85,B 0,C 180,E1 -12009.866,E2 -12009.866} C_VEL
LIN {X 0,Y 383.02,Z 179.777,A -85,B 0,C 180,E1 -12012.579,E2 -12012.579} C_VEL
LIN {X 0,Y 382.996,Z 179.775,A -85,B 0,C 180,E1 -12015.789,E2 -12015.789} C_VEL
LIN {X 0,Y 382.986,Z 179.78,A -85,B 0,C 180,E1 -12018.796,E2 -12018.796} C_VEL
LIN {X 0,Y 382.992,Z 179.777,A -85,B 0,C 180,E1 -12022.097,E2 -12022.097} C_VEL
LIN {X 0,Y 383.015,Z 179.772,A -85,B 0,C 180,E1 -12025.332,E2 -12025.332} C_VEL
LIN {X 0,Y 382.981,Z 179.777,A -85,B 0,C 180,E1 -12029.081,E2 -12029.081} C_VEL
LIN {X 0,Y 383.055,Z 179.768,A -85,B 0,C 180,E1 -12032.698,E2 -12032.698} C_VEL
LIN {X 0,Y 383.048,Z 179.768,A -85,B 0,C 180,E1 -12035.039,E2 -12035.039} C_VEL
LIN {X 0,Y 382.99,Z 179.776,A -85,B 0,C 180,E1 -12038.469,E2 -12038.469} C_VEL
LIN {X 0,Y 383.087,Z 179.767,A -85,B 0,C 180,E1 -12041.828,E2 -12041.828} C_VEL
LIN {X 0,Y 383.108,Z 179.763,A -85,B 0,C 180,E1 -12045.118,E2 -12045.118} C_VEL
LIN {X 0,Y 383.093,Z 179.762,A -85,B 0,C 180,E1 -12048.358,E2 -12048.358} C_VEL
LIN {X 0,Y 383.212,Z 179.747,A -85,B 0,C 180,E1 -12052.028,E2 -12052.028} C_VEL
LIN {X 0,Y 383.179,Z 179.754,A -85,B 0,C 180,E1 -12054.738,E2 -12054.738} C_VEL
LIN {X 0,Y 383.383,Z 179.726,A -85,B 0,C 180,E1 -12057.899,E2 -12057.899} C_VEL
LIN {X 0,Y 383.518,Z 179.71,A -85,B 0,C 180,E1 -12060,E2 -12060} C_VEL
LIN {X 0,Y 383.24,Z 179.746,A -85,B 0,C 180,E1 -12063.154,E2 -12063.154} C_VEL
LIN {X 0,Y 383.218,Z 179.748,A -85,B 0,C 180,E1 -12066.545,E2 -12066.545} C_VEL
LIN {X 0,Y 383.139,Z 179.756,A -85,B 0,C 180,E1 -12069.502,E2 -12069.502} C_VEL
LIN {X 0,Y 383.123,Z 179.759,A -85,B 0,C 180,E1 -12073.536,E2 -12073.536} C_VEL
LIN {X 0,Y 383.093,Z 179.763,A -85,B 0,C 180,E1 -12077.455,E2 -12077.455} C_VEL
LIN {X 0,Y 383.027,Z 179.771,A -85,B 0,C 180,E1 -12080.647,E2 -12080.647} C_VEL
LIN {X 0,Y 383.031,Z 179.776,A -85,B 0,C 180,E1 -12083.808,E2 -12083.808} C_VEL
LIN {X 0,Y 383.078,Z 179.767,A -85,B 0,C 180,E1 -12086.124,E2 -12086.124} C_VEL
LIN {X 0,Y 382.991,Z 179.78,A -85,B 0,C 180,E1 -12089.7,E2 -12089.7} C_VEL
LIN {X 0,Y 383.001,Z 179.779,A -85,B 0,C 180,E1 -12093.401,E2 -12093.401} C_VEL
LIN {X 0,Y 383.028,Z 179.771,A -85,B 0,C 180,E1 -12096.164,E2 -12096.164} C_VEL
LIN {X 0,Y 382.999,Z 179.774,A -85,B 0,C 180,E1 -12099.96,E2 -12099.96} C_VEL
LIN {X 0,Y 383.004,Z 179.777,A -85,B 0,C 180,E1 -12102.779,E2 -12102.779} C_VEL
LIN {X 0,Y 382.997,Z 179.775,A -85,B 0,C 180,E1 -12105.79,E2 -12105.79} C_VEL
LIN {X 0,Y 382.988,Z 179.781,A -85,B 0,C 180,E1 -12108.796,E2 -12108.796} C_VEL
LIN {X 0,Y 382.991,Z 179.777,A -85,B 0,C 180,E1 -12112.098,E2 -12112.098} C_VEL
LIN {X 0,Y 382.941,Z 180.244,A -85,B 0,C 180,E1 -12114.036,E2 -12114.036} C_VEL
LIN {X 0,Y 382.882,Z 183.196,A -85,B 0,C 180,E1 -12116.588,E2 -12116.588} C_VEL
LIN {X 0,Y 382.755,Z 186.768,A -85,B 0,C 180,E1 -12119.655,E2 -12119.655} C_VEL
LIN {X 0,Y 382.548,Z 190.411,A -85,B 0,C 180,E1 -12122.659,E2 -12122.659} C_VEL
LIN {X 0,Y 382.35,Z 194.803,A -85,B 0,C 180,E1 -12126.148,E2 -12126.148} C_VEL
LIN {X 0,Y 382.165,Z 199.465,A -85,B 0,C 180,E1 -12129.701,E2 -12129.701} C_VEL
LIN {X 0,Y 382.095,Z 201.562,A -85,B 0,C 180,E1 -12131.149,E2 -12131.149} C_VEL
LIN {X 0,Y 385.374,Z 214.671,A -85,B 0,C 180,E1 -12131.784,E2 -12131.784} C_VEL
LIN {X 0,Y 387.864,Z 227.463,A -85,B 0,C 180,E1 -12132.586,E2 -12132.586} C_VEL
LIN {X 0,Y 387.976,Z 230.339,A -85,B 0,C 180,E1 -12132.779,E2 -12132.779} C_VEL
LIN {X 0,Y 387.108,Z 242.261,A -85,B 0,C 180,E1 -12133.656,E2 -12133.656} C_VEL
LIN {X 0,Y 386.195,Z 253.596,A -85,B 0,C 180,E1 -12134.731,E2 -12134.731} C_VEL
LIN {X 0,Y 385.552,Z 262.261,A -85,B 0,C 180,E1 -12135.754,E2 -12135.754} C_VEL
LIN {X 0,Y 384.665,Z 271.438,A -85,B 0,C 180,E1 -12137.067,E2 -12137.067} C_VEL
LIN {X 0,Y 383.917,Z 279.002,A -85,B 0,C 180,E1 -12138.383,E2 -12138.383} C_VEL
LIN {X 0,Y 383.178,Z 286.411,A -85,B 0,C 180,E1 -12139.966,E2 -12139.966} C_VEL
LIN {X 0,Y 382.534,Z 292.36,A -85,B 0,C 180,E1 -12141.548,E2 -12141.548} C_VEL
LIN {X 0,Y 382.19,Z 297.27,A -85,B 0,C 180,E1 -12143.216,E2 -12143.216} C_VEL
LIN {X 0,Y 381.965,Z 300.651,A -85,B 0,C 180,E1 -12144.722,E2 -12144.722} C_VEL
LIN {X 0,Y 381.771,Z 302.511,A -85,B 0,C 180,E1 -12145.777,E2 -12145.777} C_VEL
LIN {X 0,Y 381.706,Z 303.91,A -85,B 0,C 180,E1 -12146.834,E2 -12146.834} C_VEL
LIN {X 0,Y 381.645,Z 305.516,A -85,B 0,C 180,E1 -12148.945,E2 -12148.945} C_VEL
LIN {X 0,Y 381.641,Z 305.749,A -85,B 0,C 180,E1 -12150,E2 -12150} C_VEL
LIN {X 0,Y 381.645,Z 305.56,A -85,B 0,C 180,E1 -12151.055,E2 -12151.055} C_VEL
LIN {X 0,Y 381.705,Z 304.01,A -85,B 0,C 180,E1 -12153.167,E2 -12153.167} C_VEL
LIN {X 0,Y 381.768,Z 302.656,A -85,B 0,C 180,E1 -12154.223,E2 -12154.223} C_VEL
LIN {X 0,Y 382.029,Z 299.789,A -85,B 0,C 180,E1 -12155.807,E2 -12155.807} C_VEL
LIN {X 0,Y 382.28,Z 295.906,A -85,B 0,C 180,E1 -12157.394,E2 -12157.394} C_VEL
LIN {X 0,Y 382.698,Z 290.895,A -85,B 0,C 180,E1 -12158.981,E2 -12158.981} C_VEL
LIN {X 0,Y 383.344,Z 284.582,A -85,B 0,C 180,E1 -12160.564,E2 -12160.564} C_VEL
LIN {X 0,Y 384.101,Z 276.681,A -85,B 0,C 180,E1 -12162.147,E2 -12162.147} C_VEL
LIN {X 0,Y 385.117,Z 266.849,A -85,B 0,C 180,E1 -12163.724,E2 -12163.724} C_VEL
LIN {X 0,Y 386.038,Z 256.55,A -85,B 0,C 180,E1 -12165.034,E2 -12165.034} C_VEL
LIN {X 0,Y 386.904,Z 244.888,A -85,B 0,C 180,E1 -12166.218,E2 -12166.218} C_VEL
LIN {X 0,Y 387.819,Z 234.199,A -85,B 0,C 180,E1 -12167.061,E2 -12167.061} C_VEL
LIN {X 0,Y 387.978,Z 228.143,A -85,B 0,C 180,E1 -12167.467,E2 -12167.467} C_VEL
LIN {X 0,Y 385.638,Z 215.926,A -85,B 0,C 180,E1 -12168.247,E2 -12168.247} C_VEL
LIN {X 0,Y 382.425,Z 203.154,A -85,B 0,C 180,E1 -12168.888,E2 -12168.888} C_VEL
LIN {X 0,Y 382.326,Z 202.822,A -85,B 0,C 180,E1 -12168.903,E2 -12168.903} C_VEL
LIN {X 0,Y 381.642,Z 201.577,A -85,B 0,C 180,E1 -12169.063,E2 -12169.063} C_VEL
LIN {X 0,Y 379.901,Z 200.708,A -85,B 0,C 180,E1 -12169.645,E2 -12169.645} C_VEL
LIN {X 0,Y 377.639,Z 199.483,A -85,B 0,C 180,E1 -12170.745,E2 -12170.745} C_VEL
LIN {X 0,Y 376.268,Z 198.68,A -85,B 0,C 180,E1 -12171.756,E2 -12171.756} C_VEL
LIN {X 0,Y 375.264,Z 196.253,A -85,B 0,C 180,E1 -12173.452,E2 -12173.452} C_VEL
LIN {X 0,Y 375.436,Z 192.194,A -85,B 0,C 180,E1 -12176.697,E2 -12176.697} C_VEL
LIN {X 0,Y 375.719,Z 187.805,A -85,B 0,C 180,E1 -12180.335,E2 -12180.335} C_VEL
LIN {X 0,Y 375.89,Z 183.44,A -85,B 0,C 180,E1 -12184.119,E2 -12184.119} C_VEL
LIN {X 0,Y 375.884,Z 180.665,A -85,B 0,C 180,E1 -12186.749,E2 -12186.749} C_VEL
LIN {X 0,Y 375.939,Z 180.654,A -85,B 0,C 180,E1 -12189.961,E2 -12189.961} C_VEL
LIN {X 0,Y 375.93,Z 180.656,A -85,B 0,C 180,E1 -12193.766,E2 -12193.766} C_VEL
LIN {X 0,Y 375.936,Z 180.658,A -85,B 0,C 180,E1 -12196.811,E2 -12196.811} C_VEL
LIN {X 0,Y 375.948,Z 180.655,A -85,B 0,C 180,E1 -12200.535,E2 -12200.535} C_VEL
LIN {X 0,Y 375.962,Z 180.651,A -85,B 0,C 180,E1 -12203.496,E2 -12203.496} C_VEL
LIN {X 0,Y 375.959,Z 180.651,A -85,B 0,C 180,E1 -12205.888,E2 -12205.888} C_VEL
LIN {X 0,Y 375.966,Z 180.65,A -85,B 0,C 180,E1 -12209.687,E2 -12209.687} C_VEL
LIN {X 0,Y 376.021,Z 180.643,A -85,B 0,C 180,E1 -12213.348,E2 -12213.348} C_VEL
LIN {X 0,Y 375.998,Z 180.647,A -85,B 0,C 180,E1 -12216.888,E2 -12216.888} C_VEL
LIN {X 0,Y 375.999,Z 180.649,A -85,B 0,C 180,E1 -12220.339,E2 -12220.339} C_VEL
LIN {X 0,Y 376.03,Z 180.647,A -85,B 0,C 180,E1 -12223.719,E2 -12223.719} C_VEL
LIN {X 0,Y 376.104,Z 180.633,A -85,B 0,C 180,E1 -12227.042,E2 -12227.042} C_VEL
LIN {X 0,Y 376.113,Z 180.632,A -85,B 0,C 180,E1 -12230.318,E2 -12230.318} C_VEL
LIN {X 0,Y 376.2,Z 180.626,A -85,B 0,C 180,E1 -12233.564,E2 -12233.564} C_VEL
LIN {X 0,Y 376.351,Z 180.603,A -85,B 0,C 180,E1 -12237.86,E2 -12237.86} C_VEL
LIN {X 0,Y 376.49,Z 180.585,A -85,B 0,C 180,E1 -12240,E2 -12240} C_VEL
LIN {X 0,Y 376.181,Z 180.628,A -85,B 0,C 180,E1 -12243.213,E2 -12243.213} C_VEL
LIN {X 0,Y 376.2,Z 180.622,A -85,B 0,C 180,E1 -12246.436,E2 -12246.436} C_VEL
LIN {X 0,Y 376.115,Z 180.631,A -85,B 0,C 180,E1 -12249.682,E2 -12249.682} C_VEL
LIN {X 0,Y 376.091,Z 180.635,A -85,B 0,C 180,E1 -12253.658,E2 -12253.658} C_VEL
LIN {X 0,Y 376.045,Z 180.64,A -85,B 0,C 180,E1 -12257.607,E2 -12257.607} C_VEL
LIN {X 0,Y 375.979,Z 180.65,A -85,B 0,C 180,E1 -12260.832,E2 -12260.832} C_VEL
LIN {X 0,Y 375.989,Z 180.652,A -85,B 0,C 180,E1 -12264.282,E2 -12264.282} C_VEL
LIN {X 0,Y 376.021,Z 180.644,A -85,B 0,C 180,E1 -12266.652,E2 -12266.652} C_VEL
LIN {X 0,Y 375.966,Z 180.652,A -85,B 0,C 180,E1 -12270.313,E2 -12270.313} C_VEL
LIN {X 0,Y 375.961,Z 180.653,A -85,B 0,C 180,E1 -12274.111,E2 -12274.111} C_VEL
LIN {X 0,Y 375.951,Z 180.652,A -85,B 0,C 180,E1 -12276.742,E2 -12276.742} C_VEL
LIN {X 0,Y 375.98,Z 180.65,A -85,B 0,C 180,E1 -12279.969,E2 -12279.969} C_VEL
LIN {X 0,Y 375.931,Z 180.659,A -85,B 0,C 180,E1 -12283.766,E2 -12283.766} C_VEL
LIN {X 0,Y 375.982,Z 180.714,A -85,B 0,C 180,E1 -12287.264,E2 -12287.264} C_VEL
LIN {X 0,Y 376.873,Z 185.793,A -85,B 0,C 180,E1 -12290.651,E2 -12290.651} C_VEL
LIN {X 0,Y 377.397,Z 190.205,A -85,B 0,C 180,E1 -12293.422,E2 -12293.422} C_VEL
LIN {X 0,Y 377.296,Z 194.614,A -85,B 0,C 180,E1 -12296.026,E2 -12296.026} C_VEL
LIN {X 0,Y 376.875,Z 200.003,A -85,B 0,C 180,E1 -12299.072,E2 -12299.072} C_VEL
LIN {X 0,Y 376.277,Z 206.766,A -85,B 0,C 180,E1 -12302.767,E2 -12302.767} C_VEL
LIN {X 0,Y 375.777,Z 213.556,A -85,B 0,C 180,E1 -12306.41,E2 -12306.41} C_VEL
LIN {X 0,Y 375.479,Z 219.142,A -85,B 0,C 180,E1 -12309.37,E2 -12309.37} C_VEL
LIN {X 0,Y 375.329,Z 221.798,A -85,B 0,C 180,E1 -12310.712,E2 -12310.712} C_VEL
LIN {X 0,Y 377.876,Z 234.853,A -85,B 0,C 180,E1 -12311.284,E2 -12311.284} C_VEL
LIN {X 0,Y 379.851,Z 247.996,A -85,B 0,C 180,E1 -12312.066,E2 -12312.066} C_VEL
LIN {X 0,Y 380.591,Z 254.203,A -85,B 0,C 180,E1 -12312.51,E2 -12312.51} C_VEL
LIN {X 0,Y 379.665,Z 266.459,A -85,B 0,C 180,E1 -12313.464,E2 -12313.464} C_VEL
LIN {X 0,Y 378.563,Z 278.262,A -85,B 0,C 180,E1 -12314.66,E2 -12314.66} C_VEL
LIN {X 0,Y 377.625,Z 288.748,A -85,B 0,C 180,E1 -12315.998,E2 -12315.998} C_VEL
LIN {X 0,Y 376.784,Z 297.236,A -85,B 0,C 180,E1 -12317.34,E2 -12317.34} C_VEL
LIN {X 0,Y 375.956,Z 305.518,A -85,B 0,C 180,E1 -12318.953,E2 -12318.953} C_VEL
LIN {X 0,Y 375.358,Z 312.197,A -85,B 0,C 180,E1 -12320.57,E2 -12320.57} C_VEL
LIN {X 0,Y 374.891,Z 318.311,A -85,B 0,C 180,E1 -12322.459,E2 -12322.459} C_VEL
LIN {X 0,Y 374.632,Z 321.81,A -85,B 0,C 180,E1 -12323.863,E2 -12323.863} C_VEL
LIN {X 0,Y 374.569,Z 325.223,A -85,B 0,C 180,E1 -12325.696,E2 -12325.696} C_VEL
LIN {X 0,Y 374.457,Z 327.618,A -85,B 0,C 180,E1 -12327.849,E2 -12327.849} C_VEL
LIN {X 0,Y 374.491,Z 328.228,A -85,B 0,C 180,E1 -12328.924,E2 -12328.924} C_VEL
LIN {X 0,Y 374.508,Z 328.445,A -85,B 0,C 180,E1 -12330,E2 -12330} C_VEL
LIN {X 0,Y 374.491,Z 328.228,A -85,B 0,C 180,E1 -12331.075,E2 -12331.075} C_VEL
LIN {X 0,Y 374.462,Z 326.62,A -85,B 0,C 180,E1 -12333.227,E2 -12333.227} C_VEL
LIN {X 0,Y 374.568,Z 325.224,A -85,B 0,C 180,E1 -12334.304,E2 -12334.304} C_VEL
LIN {X 0,Y 374.664,Z 321.699,A -85,B 0,C 180,E1 -12336.183,E2 -12336.183} C_VEL
LIN {X 0,Y 374.981,Z 316.708,A -85,B 0,C 180,E1 -12338.08,E2 -12338.08} C_VEL
LIN {X 0,Y 375.46,Z 311.175,A -85,B 0,C 180,E1 -12339.698,E2 -12339.698} C_VEL
LIN {X 0,Y 376.048,Z 304.268,A -85,B 0,C 180,E1 -12341.317,E2 -12341.317} C_VEL
LIN {X 0,Y 376.968,Z 295.634,A -85,B 0,C 180,E1 -12342.927,E2 -12342.927} C_VEL
LIN {X 0,Y 377.938,Z 285.725,A -85,B 0,C 180,E1 -12344.412,E2 -12344.412} C_VEL
LIN {X 0,Y 378.771,Z 275.879,A -85,B 0,C 180,E1 -12345.607,E2 -12345.607} C_VEL
LIN {X 0,Y 379.757,Z 264.887,A -85,B 0,C 180,E1 -12346.669,E2 -12346.669} C_VEL
LIN {X 0,Y 380.548,Z 254.156,A -85,B 0,C 180,E1 -12347.491,E2 -12347.491} C_VEL
LIN {X 0,Y 379.032,Z 242.016,A -85,B 0,C 180,E1 -12348.309,E2 -12348.309} C_VEL
LIN {X 0,Y 376.783,Z 228.92,A -85,B 0,C 180,E1 -12348.996,E2 -12348.996} C_VEL
LIN {X 0,Y 375.329,Z 221.634,A -85,B 0,C 180,E1 -12349.306,E2 -12349.306} C_VEL
LIN {X 0,Y 375.736,Z 214.421,A -85,B 0,C 180,E1 -12353.128,E2 -12353.128} C_VEL
LIN {X 0,Y 376.202,Z 207.853,A -85,B 0,C 180,E1 -12356.638,E2 -12356.638} C_VEL
LIN {X 0,Y 376.883,Z 199.965,A -85,B 0,C 180,E1 -12360.93,E2 -12360.93} C_VEL
LIN {X 0,Y 377.285,Z 194.568,A -85,B 0,C 180,E1 -12363.975,E2 -12363.975} C_VEL
LIN {X 0,Y 377.397,Z 190.166,A -85,B 0,C 180,E1 -12366.577,E2 -12366.577} C_VEL
LIN {X 0,Y 376.876,Z 185.771,A -85,B 0,C 180,E1 -12369.348,E2 -12369.348} C_VEL
LIN {X 0,Y 375.968,Z 180.656,A -85,B 0,C 180,E1 -12372.863,E2 -12372.863} C_VEL
LIN {X 0,Y 375.933,Z 180.659,A -85,B 0,C 180,E1 -12376.81,E2 -12376.81} C_VEL
LIN {X 0,Y 375.945,Z 180.659,A -85,B 0,C 180,E1 -12380.535,E2 -12380.535} C_VEL
LIN {X 0,Y 375.96,Z 180.651,A -85,B 0,C 180,E1 -12383.496,E2 -12383.496} C_VEL
LIN {X 0,Y 375.958,Z 180.653,A -85,B 0,C 180,E1 -12385.888,E2 -12385.888} C_VEL
LIN {X 0,Y 375.963,Z 180.653,A -85,B 0,C 180,E1 -12389.687,E2 -12389.687} C_VEL
LIN {X 0,Y 376.018,Z 180.645,A -85,B 0,C 180,E1 -12393.348,E2 -12393.348} C_VEL
LIN {X 0,Y 375.977,Z 180.648,A -85,B 0,C 180,E1 -12396.887,E2 -12396.887} C_VEL
LIN {X 0,Y 375.996,Z 180.647,A -85,B 0,C 180,E1 -12400.339,E2 -12400.339} C_VEL
LIN {X 0,Y 376.027,Z 180.647,A -85,B 0,C 180,E1 -12403.719,E2 -12403.719} C_VEL
LIN {X 0,Y 376.101,Z 180.636,A -85,B 0,C 180,E1 -12407.042,E2 -12407.042} C_VEL
LIN {X 0,Y 376.11,Z 180.632,A -85,B 0,C 180,E1 -12410.318,E2 -12410.318} C_VEL
LIN {X 0,Y 376.197,Z 180.623,A -85,B 0,C 180,E1 -12413.564,E2 -12413.564} C_VEL
LIN {X 0,Y 376.349,Z 180.602,A -85,B 0,C 180,E1 -12417.86,E2 -12417.86} C_VEL
LIN {X 0,Y 376.487,Z 180.585,A -85,B 0,C 180,E1 -12420,E2 -12420} C_VEL
LIN {X 0,Y 376.178,Z 180.625,A -85,B 0,C 180,E1 -12423.213,E2 -12423.213} C_VEL
LIN {X 0,Y 376.188,Z 180.626,A -85,B 0,C 180,E1 -12426.53,E2 -12426.53} C_VEL
LIN {X 0,Y 376.11,Z 180.632,A -85,B 0,C 180,E1 -12429.682,E2 -12429.682} C_VEL
LIN {X 0,Y 376.087,Z 180.636,A -85,B 0,C 180,E1 -12433.658,E2 -12433.658} C_VEL
LIN {X 0,Y 376.042,Z 180.642,A -85,B 0,C 180,E1 -12437.608,E2 -12437.608} C_VEL
LIN {X 0,Y 375.976,Z 180.649,A -85,B 0,C 180,E1 -12440.832,E2 -12440.832} C_VEL
LIN {X 0,Y 375.992,Z 180.649,A -85,B 0,C 180,E1 -12444.282,E2 -12444.282} C_VEL
LIN {X 0,Y 376.018,Z 180.643,A -85,B 0,C 180,E1 -12446.652,E2 -12446.652} C_VEL
LIN {X 0,Y 375.963,Z 180.651,A -85,B 0,C 180,E1 -12450.313,E2 -12450.313} C_VEL
LIN {X 0,Y 375.958,Z 180.652,A -85,B 0,C 180,E1 -12454.112,E2 -12454.112} C_VEL
LIN {X 0,Y 375.95,Z 180.653,A -85,B 0,C 180,E1 -12456.742,E2 -12456.742} C_VEL
LIN {X 0,Y 375.979,Z 180.648,A -85,B 0,C 180,E1 -12459.97,E2 -12459.97} C_VEL
LIN {X 0,Y 375.929,Z 180.655,A -85,B 0,C 180,E1 -12463.766,E2 -12463.766} C_VEL
LIN {X 0,Y 375.934,Z 180.66,A -85,B 0,C 180,E1 -12466.811,E2 -12466.811} C_VEL
LIN {X 0,Y 375.959,Z 180.655,A -85,B 0,C 180,E1 -12470.538,E2 -12470.538} C_VEL
LIN {X 0,Y 375.873,Z 180.668,A -85,B 0,C 180,E1 -12473.515,E2 -12473.515} C_VEL
LIN {X 0,Y 375.869,Z 183.319,A -85,B 0,C 180,E1 -12475.88,E2 -12475.88} C_VEL
LIN {X 0,Y 375.718,Z 187.693,A -85,B 0,C 180,E1 -12479.666,E2 -12479.666} C_VEL
LIN {X 0,Y 375.439,Z 192.052,A -85,B 0,C 180,E1 -12483.304,E2 -12483.304} C_VEL
LIN {X 0,Y 375.283,Z 196.475,A -85,B 0,C 180,E1 -12486.842,E2 -12486.842} C_VEL
LIN {X 0,Y 375.051,Z 201.646,A -85,B 0,C 180,E1 -12490.777,E2 -12490.777} C_VEL
LIN {X 0,Y 378.285,Z 214.503,A -85,B 0,C 180,E1 -12491.411,E2 -12491.411} C_VEL
LIN {X 0,Y 380.693,Z 226.73,A -85,B 0,C 180,E1 -12492.188,E2 -12492.188} C_VEL
LIN {X 0,Y 381.195,Z 230.852,A -85,B 0,C 180,E1 -12492.483,E2 -12492.483} C_VEL
LIN {X 0,Y 380.311,Z 242.479,A -85,B 0,C 180,E1 -12493.356,E2 -12493.356} C_VEL
LIN {X 0,Y 379.343,Z 253.828,A -85,B 0,C 180,E1 -12494.45,E2 -12494.45} C_VEL
LIN {X 0,Y 378.695,Z 262.477,A -85,B 0,C 180,E1 -12495.491,E2 -12495.491} C_VEL
LIN {X 0,Y 377.743,Z 271.655,A -85,B 0,C 180,E1 -12496.826,E2 -12496.826} C_VEL
LIN {X 0,Y 376.971,Z 279.217,A -85,B 0,C 180,E1 -12498.166,E2 -12498.166} C_VEL
LIN {X 0,Y 376.196,Z 286.626,A -85,B 0,C 180,E1 -12499.777,E2 -12499.777} C_VEL
LIN {X 0,Y 375.517,Z 292.574,A -85,B 0,C 180,E1 -12501.389,E2 -12501.389} C_VEL
LIN {X 0,Y 375.129,Z 297.763,A -85,B 0,C 180,E1 -12503.195,E2 -12503.195} C_VEL
LIN {X 0,Y 374.892,Z 300.865,A -85,B 0,C 180,E1 -12504.622,E2 -12504.622} C_VEL
LIN {X 0,Y 374.703,Z 302.725,A -85,B 0,C 180,E1 -12505.698,E2 -12505.698} C_VEL
LIN {X 0,Y 374.614,Z 304.123,A -85,B 0,C 180,E1 -12506.774,E2 -12506.774} C_VEL
LIN {X 0,Y 374.562,Z 305.729,A -85,B 0,C 180,E1 -12508.925,E2 -12508.925} C_VEL
LIN {X 0,Y 374.556,Z 305.961,A -85,B 0,C 180,E1 -12510,E2 -12510} C_VEL
LIN {X 0,Y 374.563,Z 305.772,A -85,B 0,C 180,E1 -12511.075,E2 -12511.075} C_VEL
LIN {X 0,Y 374.612,Z 304.223,A -85,B 0,C 180,E1 -12513.227,E2 -12513.227} C_VEL
LIN {X 0,Y 374.7,Z 302.868,A -85,B 0,C 180,E1 -12514.303,E2 -12514.303} C_VEL
LIN {X 0,Y 374.969,Z 300.001,A -85,B 0,C 180,E1 -12515.917,E2 -12515.917} C_VEL
LIN {X 0,Y 375.238,Z 296.118,A -85,B 0,C 180,E1 -12517.534,E2 -12517.534} C_VEL
LIN {X 0,Y 375.676,Z 291.106,A -85,B 0,C 180,E1 -12519.15,E2 -12519.15} C_VEL
LIN {X 0,Y 376.358,Z 284.793,A -85,B 0,C 180,E1 -12520.763,E2 -12520.763} C_VEL
LIN {X 0,Y 377.161,Z 276.892,A -85,B 0,C 180,E1 -12522.374,E2 -12522.374} C_VEL
LIN {X 0,Y 378.228,Z 267.058,A -85,B 0,C 180,E1 -12523.979,E2 -12523.979} C_VEL
LIN {X 0,Y 379.158,Z 256.76,A -85,B 0,C 180,E1 -12525.313,E2 -12525.313} C_VEL
LIN {X 0,Y 380.087,Z 245.096,A -85,B 0,C 180,E1 -12526.517,E2 -12526.517} C_VEL
LIN {X 0,Y 381.059,Z 233.149,A -85,B 0,C 180,E1 -12527.464,E2 -12527.464} C_VEL
LIN {X 0,Y 381.121,Z 228.822,A -85,B 0,C 180,E1 -12527.762,E2 -12527.762} C_VEL
LIN {X 0,Y 378.568,Z 215.847,A -85,B 0,C 180,E1 -12528.613,E2 -12528.613} C_VEL
LIN {X 0,Y 375.292,Z 203.009,A -85,B 0,C 180,E1 -12529.272,E2 -12529.272} C_VEL
LIN {X 0,Y 375.059,Z 201.59,A -85,B 0,C 180,E1 -12529.356,E2 -12529.356} C_VEL
LIN {X 0,Y 375.251,Z 196.623,A -85,B 0,C 180,E1 -12533.16,E2 -12533.16} C_VEL
LIN {X 0,Y 375.264,Z 196.253,A -85,B 0,C 180,E1 -12533.452,E2 -12533.452} C_VEL
LIN {X 0,Y 374.597,Z 195.221,A -85,B 0,C 180,E1 -12534.335,E2 -12534.335} C_VEL
LIN {X 0,Y 371.803,Z 193.756,A -85,B 0,C 180,E1 -12535.779,E2 -12535.779} C_VEL
LIN {X 0,Y 369.486,Z 192.613,A -85,B 0,C 180,E1 -12536.947,E2 -12536.947} C_VEL
LIN {X 0,Y 368.548,Z 191.643,A -85,B 0,C 180,E1 -12537.846,E2 -12537.846} C_VEL
LIN {X 0,Y 368.5,Z 191.286,A -85,B 0,C 180,E1 -12538.149,E2 -12538.149} C_VEL
LIN {X 0,Y 368.692,Z 187.989,A -85,B 0,C 180,E1 -12540.976,E2 -12540.976} C_VEL
LIN {X 0,Y 368.819,Z 185.043,A -85,B 0,C 180,E1 -12543.546,E2 -12543.546} C_VEL
LIN {X 0,Y 368.872,Z 182.114,A -85,B 0,C 180,E1 -12546.202,E2 -12546.202} C_VEL
LIN {X 0,Y 368.841,Z 181.542,A -85,B 0,C 180,E1 -12546.843,E2 -12546.843} C_VEL
LIN {X 0,Y 368.884,Z 181.532,A -85,B 0,C 180,E1 -12550.374,E2 -12550.374} C_VEL
LIN {X 0,Y 368.883,Z 181.534,A -85,B 0,C 180,E1 -12553.616,E2 -12553.616} C_VEL
LIN {X 0,Y 368.887,Z 181.534,A -85,B 0,C 180,E1 -12556.696,E2 -12556.696} C_VEL
LIN {X 0,Y 368.91,Z 181.529,A -85,B 0,C 180,E1 -12559.644,E2 -12559.644} C_VEL
LIN {X 0,Y 368.899,Z 181.533,A -85,B 0,C 180,E1 -12563.145,E2 -12563.145} C_VEL
LIN {X 0,Y 368.896,Z 181.535,A -85,B 0,C 180,E1 -12566.462,E2 -12566.462} C_VEL
LIN {X 0,Y 368.931,Z 181.528,A -85,B 0,C 180,E1 -12569.046,E2 -12569.046} C_VEL
LIN {X 0,Y 368.964,Z 181.524,A -85,B 0,C 180,E1 -12572.796,E2 -12572.796} C_VEL
LIN {X 0,Y 368.947,Z 181.529,A -85,B 0,C 180,E1 -12576.113,E2 -12576.113} C_VEL
LIN {X 0,Y 368.938,Z 181.53,A -85,B 0,C 180,E1 -12579.947,E2 -12579.947} C_VEL
LIN {X 0,Y 368.977,Z 181.522,A -85,B 0,C 180,E1 -12583.399,E2 -12583.399} C_VEL
LIN {X 0,Y 369.059,Z 181.51,A -85,B 0,C 180,E1 -12586.79,E2 -12586.79} C_VEL
LIN {X 0,Y 369.063,Z 181.511,A -85,B 0,C 180,E1 -12590.132,E2 -12590.132} C_VEL
LIN {X 0,Y 369.16,Z 181.504,A -85,B 0,C 180,E1 -12593.441,E2 -12593.441} C_VEL
LIN {X 0,Y 369.316,Z 181.48,A -85,B 0,C 180,E1 -12597.819,E2 -12597.819} C_VEL
LIN {X 0,Y 369.46,Z 181.461,A -85,B 0,C 180,E1 -12600,E2 -12600} C_VEL
LIN {X 0,Y 369.317,Z 181.478,A -85,B 0,C 180,E1 -12602.181,E2 -12602.181} C_VEL
LIN {X 0,Y 369.161,Z 181.5,A -85,B 0,C 180,E1 -12606.559,E2 -12606.559} C_VEL
LIN {X 0,Y 369.065,Z 181.509,A -85,B 0,C 180,E1 -12609.868,E2 -12609.868} C_VEL
LIN {X 0,Y 369.039,Z 181.513,A -85,B 0,C 180,E1 -12613.773,E2 -12613.773} C_VEL
LIN {X 0,Y 369.002,Z 181.518,A -85,B 0,C 180,E1 -12617.768,E2 -12617.768} C_VEL
LIN {X 0,Y 368.91,Z 181.529,A -85,B 0,C 180,E1 -12621.221,E2 -12621.221} C_VEL
LIN {X 0,Y 368.955,Z 181.524,A -85,B 0,C 180,E1 -12624.776,E2 -12624.776} C_VEL
LIN {X 0,Y 368.964,Z 181.522,A -85,B 0,C 180,E1 -12627.203,E2 -12627.203} C_VEL
LIN {X 0,Y 368.93,Z 181.526,A -85,B 0,C 180,E1 -12630.954,E2 -12630.954} C_VEL
LIN {X 0,Y 368.929,Z 181.527,A -85,B 0,C 180,E1 -12635.001,E2 -12635.001} C_VEL
LIN {X 0,Y 368.88,Z 181.533,A -85,B 0,C 180,E1 -12638.634,E2 -12638.634} C_VEL
LIN {X 0,Y 368.882,Z 181.533,A -85,B 0,C 180,E1 -12642.009,E2 -12642.009} C_VEL
LIN {X 0,Y 368.881,Z 181.538,A -85,B 0,C 180,E1 -12645.176,E2 -12645.176} C_VEL
LIN {X 0,Y 368.925,Z 181.617,A -85,B 0,C 180,E1 -12646.943,E2 -12646.943} C_VEL
LIN {X 0,Y 369.844,Z 186.764,A -85,B 0,C 180,E1 -12650.463,E2 -12650.463} C_VEL
LIN {X 0,Y 370.326,Z 190.459,A -85,B 0,C 180,E1 -12652.851,E2 -12652.851} C_VEL
LIN {X 0,Y 370.368,Z 194.47,A -85,B 0,C 180,E1 -12655.3,E2 -12655.3} C_VEL
LIN {X 0,Y 370.002,Z 198.872,A -85,B 0,C 180,E1 -12657.87,E2 -12657.87} C_VEL
LIN {X 0,Y 369.454,Z 204.513,A -85,B 0,C 180,E1 -12661.05,E2 -12661.05} C_VEL
LIN {X 0,Y 368.946,Z 210.957,A -85,B 0,C 180,E1 -12664.621,E2 -12664.621} C_VEL
LIN {X 0,Y 368.515,Z 217.486,A -85,B 0,C 180,E1 -12668.168,E2 -12668.168} C_VEL
LIN {X 0,Y 368.277,Z 221.592,A -85,B 0,C 180,E1 -12670.328,E2 -12670.328} C_VEL
LIN {X 0,Y 370.943,Z 234.892,A -85,B 0,C 180,E1 -12670.933,E2 -12670.933} C_VEL
LIN {X 0,Y 372.847,Z 247.453,A -85,B 0,C 180,E1 -12671.697,E2 -12671.697} C_VEL
LIN {X 0,Y 373.717,Z 255.588,A -85,B 0,C 180,E1 -12672.291,E2 -12672.291} C_VEL
LIN {X 0,Y 372.709,Z 267.679,A -85,B 0,C 180,E1 -12673.288,E2 -12673.288} C_VEL
LIN {X 0,Y 371.579,Z 279.228,A -85,B 0,C 180,E1 -12674.505,E2 -12674.505} C_VEL
LIN {X 0,Y 370.693,Z 288.536,A -85,B 0,C 180,E1 -12675.731,E2 -12675.731} C_VEL
LIN {X 0,Y 369.839,Z 297.024,A -85,B 0,C 180,E1 -12677.098,E2 -12677.098} C_VEL
LIN {X 0,Y 368.932,Z 305.305,A -85,B 0,C 180,E1 -12678.74,E2 -12678.74} C_VEL
LIN {X 0,Y 368.318,Z 311.984,A -85,B 0,C 180,E1 -12680.389,E2 -12680.389} C_VEL
LIN {X 0,Y 367.811,Z 318.098,A -85,B 0,C 180,E1 -12682.313,E2 -12682.313} C_VEL
LIN {X 0,Y 367.538,Z 321.943,A -85,B 0,C 180,E1 -12683.9,E2 -12683.9} C_VEL
LIN {X 0,Y 367.475,Z 325.01,A -85,B 0,C 180,E1 -12685.612,E2 -12685.612} C_VEL
LIN {X 0,Y 367.358,Z 327.405,A -85,B 0,C 180,E1 -12687.807,E2 -12687.807} C_VEL
LIN {X 0,Y 367.392,Z 328.015,A -85,B 0,C 180,E1 -12688.904,E2 -12688.904} C_VEL
LIN {X 0,Y 367.411,Z 328.232,A -85,B 0,C 180,E1 -12690,E2 -12690} C_VEL
LIN {X 0,Y 367.392,Z 328.015,A -85,B 0,C 180,E1 -12691.096,E2 -12691.096} C_VEL
LIN {X 0,Y 367.381,Z 326.407,A -85,B 0,C 180,E1 -12693.29,E2 -12693.29} C_VEL
LIN {X 0,Y 367.475,Z 325.01,A -85,B 0,C 180,E1 -12694.387,E2 -12694.387} C_VEL
LIN {X 0,Y 367.557,Z 321.88,A -85,B 0,C 180,E1 -12696.127,E2 -12696.127} C_VEL
LIN {X 0,Y 367.799,Z 318.088,A -85,B 0,C 180,E1 -12697.687,E2 -12697.687} C_VEL
LIN {X 0,Y 368.317,Z 311.972,A -85,B 0,C 180,E1 -12699.611,E2 -12699.611} C_VEL
LIN {X 0,Y 368.931,Z 305.29,A -85,B 0,C 180,E1 -12701.26,E2 -12701.26} C_VEL
LIN {X 0,Y 369.831,Z 297.005,A -85,B 0,C 180,E1 -12702.902,E2 -12702.902} C_VEL
LIN {X 0,Y 370.704,Z 288.512,A -85,B 0,C 180,E1 -12704.268,E2 -12704.268} C_VEL
LIN {X 0,Y 371.702,Z 278.018,A -85,B 0,C 180,E1 -12705.63,E2 -12705.63} C_VEL
LIN {X 0,Y 372.669,Z 267.64,A -85,B 0,C 180,E1 -12706.714,E2 -12706.714} C_VEL
LIN {X 0,Y 373.727,Z 255.539,A -85,B 0,C 180,E1 -12707.707,E2 -12707.707} C_VEL
LIN {X 0,Y 372.332,Z 243.767,A -85,B 0,C 180,E1 -12708.543,E2 -12708.543} C_VEL
LIN {X 0,Y 370.111,Z 230.42,A -85,B 0,C 180,E1 -12709.286,E2 -12709.286} C_VEL
LIN {X 0,Y 368.288,Z 221.425,A -85,B 0,C 180,E1 -12709.689,E2 -12709.689} C_VEL
LIN {X 0,Y 368.662,Z 215.319,A -85,B 0,C 180,E1 -12713.004,E2 -12713.004} C_VEL
LIN {X 0,Y 369.115,Z 208.902,A -85,B 0,C 180,E1 -12716.506,E2 -12716.506} C_VEL
LIN {X 0,Y 369.69,Z 202.153,A -85,B 0,C 180,E1 -12720.25,E2 -12720.25} C_VEL
LIN {X 0,Y 370.183,Z 196.637,A -85,B 0,C 180,E1 -12723.406,E2 -12723.406} C_VEL
LIN {X 0,Y 370.439,Z 192.227,A -85,B 0,C 180,E1 -12726.024,E2 -12726.024} C_VEL
LIN {X 0,Y 370.002,Z 187.767,A -85,B 0,C 180,E1 -12728.851,E2 -12728.851} C_VEL
LIN {X 0,Y 369.168,Z 183.04,A -85,B 0,C 180,E1 -12732.059,E2 -12732.059} C_VEL
LIN {X 0,Y 368.908,Z 181.534,A -85,B 0,C 180,E1 -12733.175,E2 -12733.175} C_VEL
LIN {X 0,Y 368.885,Z 181.538,A -85,B 0,C 180,E1 -12736.696,E2 -12736.696} C_VEL
LIN {X 0,Y 368.907,Z 181.529,A -85,B 0,C 180,E1 -12739.643,E2 -12739.643} C_VEL
LIN {X 0,Y 368.897,Z 181.531,A -85,B 0,C 180,E1 -12743.145,E2 -12743.145} C_VEL
LIN {X 0,Y 368.895,Z 181.535,A -85,B 0,C 180,E1 -12746.462,E2 -12746.462} C_VEL
LIN {X 0,Y 368.927,Z 181.527,A -85,B 0,C 180,E1 -12749.046,E2 -12749.046} C_VEL
LIN {X 0,Y 368.961,Z 181.523,A -85,B 0,C 180,E1 -12752.796,E2 -12752.796} C_VEL
LIN {X 0,Y 368.932,Z 181.53,A -85,B 0,C 180,E1 -12756.117,E2 -12756.117} C_VEL
LIN {X 0,Y 368.935,Z 181.529,A -85,B 0,C 180,E1 -12759.947,E2 -12759.947} C_VEL
LIN {X 0,Y 368.974,Z 181.525,A -85,B 0,C 180,E1 -12763.399,E2 -12763.399} C_VEL
LIN {X 0,Y 369.055,Z 181.512,A -85,B 0,C 180,E1 -12766.79,E2 -12766.79} C_VEL
LIN {X 0,Y 369.06,Z 181.51,A -85,B 0,C 180,E1 -12770.132,E2 -12770.132} C_VEL
LIN {X 0,Y 369.157,Z 181.501,A -85,B 0,C 180,E1 -12773.441,E2 -12773.441} C_VEL
LIN {X 0,Y 369.313,Z 181.479,A -85,B 0,C 180,E1 -12777.819,E2 -12777.819} C_VEL
LIN {X 0,Y 369.456,Z 181.461,A -85,B 0,C 180,E1 -12780,E2 -12780} C_VEL
LIN {X 0,Y 369.313,Z 181.48,A -85,B 0,C 180,E1 -12782.181,E2 -12782.181} C_VEL
LIN {X 0,Y 369.157,Z 181.504,A -85,B 0,C 180,E1 -12786.559,E2 -12786.559} C_VEL
LIN {X 0,Y 369.06,Z 181.511,A -85,B 0,C 180,E1 -12789.869,E2 -12789.869} C_VEL
LIN {X 0,Y 369.035,Z 181.515,A -85,B 0,C 180,E1 -12793.772,E2 -12793.772} C_VEL
LIN {X 0,Y 368.999,Z 181.521,A -85,B 0,C 180,E1 -12797.769,E2 -12797.769} C_VEL
LIN {X 0,Y 368.927,Z 181.527,A -85,B 0,C 180,E1 -12801.22,E2 -12801.22} C_VEL
LIN {X 0,Y 368.956,Z 181.523,A -85,B 0,C 180,E1 -12804.776,E2 -12804.776} C_VEL
LIN {X 0,Y 368.961,Z 181.524,A -85,B 0,C 180,E1 -12807.204,E2 -12807.204} C_VEL
LIN {X 0,Y 368.928,Z 181.528,A -85,B 0,C 180,E1 -12810.954,E2 -12810.954} C_VEL
LIN {X 0,Y 368.927,Z 181.529,A -85,B 0,C 180,E1 -12815.002,E2 -12815.002} C_VEL
LIN {X 0,Y 368.879,Z 181.534,A -85,B 0,C 180,E1 -12818.635,E2 -12818.635} C_VEL
LIN {X 0,Y 368.88,Z 181.532,A -85,B 0,C 180,E1 -12822.01,E2 -12822.01} C_VEL
LIN {X 0,Y 368.879,Z 181.536,A -85,B 0,C 180,E1 -12825.176,E2 -12825.176} C_VEL
LIN {X 0,Y 368.882,Z 181.533,A -85,B 0,C 180,E1 -12828.178,E2 -12828.178} C_VEL
LIN {X 0,Y 368.902,Z 181.53,A -85,B 0,C 180,E1 -12831.361,E2 -12831.361} C_VEL
LIN {X 0,Y 368.837,Z 181.545,A -85,B 0,C 180,E1 -12833.158,E2 -12833.158} C_VEL
LIN {X 0,Y 368.881,Z 183.455,A -85,B 0,C 180,E1 -12835.141,E2 -12835.141} C_VEL
LIN {X 0,Y 368.751,Z 186.402,A -85,B 0,C 180,E1 -12837.748,E2 -12837.748} C_VEL
LIN {X 0,Y 368.544,Z 190.768,A -85,B 0,C 180,E1 -12841.528,E2 -12841.528} C_VEL
LIN {X 0,Y 368.268,Z 195.188,A -85,B 0,C 180,E1 -12845.176,E2 -12845.176} C_VEL
LIN {X 0,Y 368.157,Z 198.161,A -85,B 0,C 180,E1 -12847.556,E2 -12847.556} C_VEL
LIN {X 0,Y 368.024,Z 201.899,A -85,B 0,C 180,E1 -12850.395,E2 -12850.395} C_VEL
LIN {X 0,Y 371.334,Z 215.084,A -85,B 0,C 180,E1 -12851.067,E2 -12851.067} C_VEL
LIN {X 0,Y 373.836,Z 227.485,A -85,B 0,C 180,E1 -12851.883,E2 -12851.883} C_VEL
LIN {X 0,Y 374.421,Z 231.34,A -85,B 0,C 180,E1 -12852.175,E2 -12852.175} C_VEL
LIN {X 0,Y 373.511,Z 242.699,A -85,B 0,C 180,E1 -12853.044,E2 -12853.044} C_VEL
LIN {X 0,Y 372.645,Z 252.997,A -85,B 0,C 180,E1 -12854.047,E2 -12854.047} C_VEL
LIN {X 0,Y 371.841,Z 262.694,A -85,B 0,C 180,E1 -12855.217,E2 -12855.217} C_VEL
LIN {X 0,Y 370.835,Z 271.871,A -85,B 0,C 180,E1 -12856.576,E2 -12856.576} C_VEL
LIN {X 0,Y 369.861,Z 280.78,A -85,B 0,C 180,E1 -12858.214,E2 -12858.214} C_VEL
LIN {X 0,Y 369.067,Z 287.952,A -85,B 0,C 180,E1 -12859.855,E2 -12859.855} C_VEL
LIN {X 0,Y 368.489,Z 292.789,A -85,B 0,C 180,E1 -12861.224,E2 -12861.224} C_VEL
LIN {X 0,Y 368.067,Z 298.242,A -85,B 0,C 180,E1 -12863.174,E2 -12863.174} C_VEL
LIN {X 0,Y 367.824,Z 301.079,A -85,B 0,C 180,E1 -12864.518,E2 -12864.518} C_VEL
LIN {X 0,Y 367.637,Z 302.938,A -85,B 0,C 180,E1 -12865.615,E2 -12865.615} C_VEL
LIN {X 0,Y 367.526,Z 304.337,A -85,B 0,C 180,E1 -12866.712,E2 -12866.712} C_VEL
LIN {X 0,Y 367.466,Z 305.942,A -85,B 0,C 180,E1 -12868.904,E2 -12868.904} C_VEL
LIN {X 0,Y 367.459,Z 306.174,A -85,B 0,C 180,E1 -12870,E2 -12870} C_VEL
LIN {X 0,Y 367.466,Z 305.985,A -85,B 0,C 180,E1 -12871.096,E2 -12871.096} C_VEL
LIN {X 0,Y 367.524,Z 304.435,A -85,B 0,C 180,E1 -12873.289,E2 -12873.289} C_VEL
LIN {X 0,Y 367.634,Z 303.079,A -85,B 0,C 180,E1 -12874.386,E2 -12874.386} C_VEL
LIN {X 0,Y 367.911,Z 300.213,A -85,B 0,C 180,E1 -12876.031,E2 -12876.031} C_VEL
LIN {X 0,Y 368.192,Z 296.33,A -85,B 0,C 180,E1 -12877.679,E2 -12877.679} C_VEL
LIN {X 0,Y 368.673,Z 291.318,A -85,B 0,C 180,E1 -12879.325,E2 -12879.325} C_VEL
LIN {X 0,Y 369.38,Z 285.004,A -85,B 0,C 180,E1 -12880.968,E2 -12880.968} C_VEL
LIN {X 0,Y 370.209,Z 277.102,A -85,B 0,C 180,E1 -12882.61,E2 -12882.61} C_VEL
LIN {X 0,Y 371.344,Z 267.268,A -85,B 0,C 180,E1 -12884.243,E2 -12884.243} C_VEL
LIN {X 0,Y 372.249,Z 257.644,A -85,B 0,C 180,E1 -12885.524,E2 -12885.524} C_VEL
LIN {X 0,Y 373.178,Z 246.725,A -85,B 0,C 180,E1 -12886.691,E2 -12886.691} C_VEL
LIN {X 0,Y 374.238,Z 234.856,A -85,B 0,C 180,E1 -12887.681,E2 -12887.681} C_VEL
LIN {X 0,Y 374.22,Z 229.441,A -85,B 0,C 180,E1 -12888.073,E2 -12888.073} C_VEL
LIN {X 0,Y 371.67,Z 216.48,A -85,B 0,C 180,E1 -12888.952,E2 -12888.952} C_VEL
LIN {X 0,Y 368.317,Z 203.47,A -85,B 0,C 180,E1 -12889.644,E2 -12889.644} C_VEL
LIN {X 0,Y 367.981,Z 201.84,A -85,B 0,C 180,E1 -12889.713,E2 -12889.713} C_VEL
LIN {X 0,Y 368.2,Z 196.986,A -85,B 0,C 180,E1 -12893.495,E2 -12893.495} C_VEL
LIN {X 0,Y 368.444,Z 192.378,A -85,B 0,C 180,E1 -12897.245,E2 -12897.245} C_VEL
LIN {X 0,Y 368.5,Z 191.286,A -85,B 0,C 180,E1 -12898.149,E2 -12898.149} C_VEL
LIN {X 0,Y 367.914,Z 190.301,A -85,B 0,C 180,E1 -12899.05,E2 -12899.05} C_VEL
LIN {X 0,Y 365.119,Z 188.971,A -85,B 0,C 180,E1 -12900.524,E2 -12900.524} C_VEL
LIN {X 0,Y 362.754,Z 187.928,A -85,B 0,C 180,E1 -12901.717,E2 -12901.717} C_VEL
LIN {X 0,Y 361.798,Z 187.029,A -85,B 0,C 180,E1 -12902.637,E2 -12902.637} C_VEL
LIN {X 0,Y 361.754,Z 186.693,A -85,B 0,C 180,E1 -12902.947,E2 -12902.947} C_VEL
LIN {X 0,Y 361.839,Z 183.731,A -85,B 0,C 180,E1 -12905.64,E2 -12905.64} C_VEL
LIN {X 0,Y 361.812,Z 182.418,A -85,B 0,C 180,E1 -12907.212,E2 -12907.212} C_VEL
LIN {X 0,Y 361.814,Z 182.414,A -85,B 0,C 180,E1 -12910.751,E2 -12910.751} C_VEL
LIN {X 0,Y 361.817,Z 182.413,A -85,B 0,C 180,E1 -12914.369,E2 -12914.369} C_VEL
LIN {X 0,Y 361.837,Z 182.411,A -85,B 0,C 180,E1 -12917.568,E2 -12917.568} C_VEL
LIN {X 0,Y 361.833,Z 182.415,A -85,B 0,C 180,E1 -12920.981,E2 -12920.981} C_VEL
LIN {X 0,Y 361.874,Z 182.411,A -85,B 0,C 180,E1 -12924.656,E2 -12924.656} C_VEL
LIN {X 0,Y 361.839,Z 182.414,A -85,B 0,C 180,E1 -12928.37,E2 -12928.37} C_VEL
LIN {X 0,Y 361.91,Z 182.405,A -85,B 0,C 180,E1 -12932.221,E2 -12932.221} C_VEL
LIN {X 0,Y 361.93,Z 182.4,A -85,B 0,C 180,E1 -12934.71,E2 -12934.71} C_VEL
LIN {X 0,Y 361.893,Z 182.407,A -85,B 0,C 180,E1 -12938.347,E2 -12938.347} C_VEL
LIN {X 0,Y 361.969,Z 182.398,A -85,B 0,C 180,E1 -12942.061,E2 -12942.061} C_VEL
LIN {X 0,Y 361.999,Z 182.393,A -85,B 0,C 180,E1 -12946.101,E2 -12946.101} C_VEL
LIN {X 0,Y 362,Z 182.392,A -85,B 0,C 180,E1 -12949.937,E2 -12949.937} C_VEL
LIN {X 0,Y 362.123,Z 182.378,A -85,B 0,C 180,E1 -12953.313,E2 -12953.313} C_VEL
LIN {X 0,Y 362.28,Z 182.356,A -85,B 0,C 180,E1 -12957.776,E2 -12957.776} C_VEL
LIN {X 0,Y 362.429,Z 182.336,A -85,B 0,C 180,E1 -12960,E2 -12960} C_VEL
LIN {X 0,Y 362.28,Z 182.355,A -85,B 0,C 180,E1 -12962.224,E2 -12962.224} C_VEL
LIN {X 0,Y 362.124,Z 182.378,A -85,B 0,C 180,E1 -12966.687,E2 -12966.687} C_VEL
LIN {X 0,Y 362.031,Z 182.386,A -85,B 0,C 180,E1 -12970.062,E2 -12970.062} C_VEL
LIN {X 0,Y 362,Z 182.39,A -85,B 0,C 180,E1 -12973.899,E2 -12973.899} C_VEL
LIN {X 0,Y 361.968,Z 182.395,A -85,B 0,C 180,E1 -12977.939,E2 -12977.939} C_VEL
LIN {X 0,Y 361.862,Z 182.408,A -85,B 0,C 180,E1 -12981.655,E2 -12981.655} C_VEL
LIN {X 0,Y 361.928,Z 182.399,A -85,B 0,C 180,E1 -12985.29,E2 -12985.29} C_VEL
LIN {X 0,Y 361.909,Z 182.405,A -85,B 0,C 180,E1 -12987.779,E2 -12987.779} C_VEL
LIN {X 0,Y 361.839,Z 182.414,A -85,B 0,C 180,E1 -12991.629,E2 -12991.629} C_VEL
LIN {X 0,Y 361.874,Z 182.408,A -85,B 0,C 180,E1 -12995.345,E2 -12995.345} C_VEL
LIN {X 0,Y 361.831,Z 182.412,A -85,B 0,C 180,E1 -12999.019,E2 -12999.019} C_VEL
LIN {X 0,Y 361.837,Z 182.411,A -85,B 0,C 180,E1 -13002.829,E2 -13002.829} C_VEL
LIN {X 0,Y 361.855,Z 182.487,A -85,B 0,C 180,E1 -13006.584,E2 -13006.584} C_VEL
LIN {X 0,Y 362.808,Z 187.721,A -85,B 0,C 180,E1 -13010.264,E2 -13010.264} C_VEL
LIN {X 0,Y 363.263,Z 191.072,A -85,B 0,C 180,E1 -13012.488,E2 -13012.488} C_VEL
LIN {X 0,Y 363.357,Z 195.413,A -85,B 0,C 180,E1 -13015.209,E2 -13015.209} C_VEL
LIN {X 0,Y 362.888,Z 200.909,A -85,B 0,C 180,E1 -13018.472,E2 -13018.472} C_VEL
LIN {X 0,Y 362.236,Z 207.508,A -85,B 0,C 180,E1 -13022.248,E2 -13022.248} C_VEL
LIN {X 0,Y 361.704,Z 214.109,A -85,B 0,C 180,E1 -13025.955,E2 -13025.955} C_VEL
LIN {X 0,Y 361.26,Z 221.029,A -85,B 0,C 180,E1 -13029.799,E2 -13029.799} C_VEL
LIN {X 0,Y 361.268,Z 221.386,A -85,B 0,C 180,E1 -13029.93,E2 -13029.93} C_VEL
LIN {X 0,Y 363.94,Z 234.813,A -85,B 0,C 180,E1 -13030.558,E2 -13030.558} C_VEL
LIN {X 0,Y 365.887,Z 247.239,A -85,B 0,C 180,E1 -13031.336,E2 -13031.336} C_VEL
LIN {X 0,Y 366.854,Z 256.71,A -85,B 0,C 180,E1 -13032.055,E2 -13032.055} C_VEL
LIN {X 0,Y 365.743,Z 268.898,A -85,B 0,C 180,E1 -13033.104,E2 -13033.104} C_VEL
LIN {X 0,Y 364.593,Z 280.153,A -85,B 0,C 180,E1 -13034.343,E2 -13034.343} C_VEL
LIN {X 0,Y 363.604,Z 290.125,A -85,B 0,C 180,E1 -13035.733,E2 -13035.733} C_VEL
LIN {X 0,Y 362.569,Z 299.794,A -85,B 0,C 180,E1 -13037.404,E2 -13037.404} C_VEL
LIN {X 0,Y 361.718,Z 307.492,A -85,B 0,C 180,E1 -13039.08,E2 -13039.08} C_VEL
LIN {X 0,Y 361.045,Z 314.593,A -85,B 0,C 180,E1 -13041.041,E2 -13041.041} C_VEL
LIN {X 0,Y 360.634,Z 319.319,A -85,B 0,C 180,E1 -13042.722,E2 -13042.722} C_VEL
LIN {X 0,Y 360.422,Z 322.932,A -85,B 0,C 180,E1 -13044.405,E2 -13044.405} C_VEL
LIN {X 0,Y 360.385,Z 324.797,A -85,B 0,C 180,E1 -13045.526,E2 -13045.526} C_VEL
LIN {X 0,Y 360.302,Z 326.194,A -85,B 0,C 180,E1 -13046.645,E2 -13046.645} C_VEL
LIN {X 0,Y 360.292,Z 327.802,A -85,B 0,C 180,E1 -13048.882,E2 -13048.882} C_VEL
LIN {X 0,Y 360.314,Z 328.019,A -85,B 0,C 180,E1 -13050,E2 -13050} C_VEL
LIN {X 0,Y 360.292,Z 327.801,A -85,B 0,C 180,E1 -13051.117,E2 -13051.117} C_VEL
LIN {X 0,Y 360.302,Z 326.194,A -85,B 0,C 180,E1 -13053.354,E2 -13053.354} C_VEL
LIN {X 0,Y 360.385,Z 324.796,A -85,B 0,C 180,E1 -13054.474,E2 -13054.474} C_VEL
LIN {X 0,Y 360.462,Z 321.983,A -85,B 0,C 180,E1 -13056.088,E2 -13056.088} C_VEL
LIN {X 0,Y 360.735,Z 317.873,A -85,B 0,C 180,E1 -13057.838,E2 -13057.838} C_VEL
LIN {X 0,Y 361.294,Z 311.757,A -85,B 0,C 180,E1 -13059.8,E2 -13059.8} C_VEL
LIN {X 0,Y 361.937,Z 305.075,A -85,B 0,C 180,E1 -13061.48,E2 -13061.48} C_VEL
LIN {X 0,Y 362.893,Z 296.789,A -85,B 0,C 180,E1 -13063.153,E2 -13063.153} C_VEL
LIN {X 0,Y 363.812,Z 288.296,A -85,B 0,C 180,E1 -13064.544,E2 -13064.544} C_VEL
LIN {X 0,Y 364.841,Z 277.801,A -85,B 0,C 180,E1 -13065.932,E2 -13065.932} C_VEL
LIN {X 0,Y 366.014,Z 265.993,A -85,B 0,C 180,E1 -13067.171,E2 -13067.171} C_VEL
LIN {X 0,Y 366.813,Z 255.461,A -85,B 0,C 180,E1 -13068.041,E2 -13068.041} C_VEL
LIN {X 0,Y 365.162,Z 242.358,A -85,B 0,C 180,E1 -13068.987,E2 -13068.987} C_VEL
LIN {X 0,Y 363.03,Z 229.825,A -85,B 0,C 180,E1 -13069.692,E2 -13069.692} C_VEL
LIN {X 0,Y 361.254,Z 221.219,A -85,B 0,C 180,E1 -13070.089,E2 -13070.089} C_VEL
LIN {X 0,Y 361.744,Z 214.034,A -85,B 0,C 180,E1 -13074.078,E2 -13074.078} C_VEL
LIN {X 0,Y 362.235,Z 207.495,A -85,B 0,C 180,E1 -13077.751,E2 -13077.751} C_VEL
LIN {X 0,Y 362.878,Z 200.851,A -85,B 0,C 180,E1 -13081.552,E2 -13081.552} C_VEL
LIN {X 0,Y 363.353,Z 195.375,A -85,B 0,C 180,E1 -13084.791,E2 -13084.791} C_VEL
LIN {X 0,Y 363.263,Z 191.023,A -85,B 0,C 180,E1 -13087.512,E2 -13087.512} C_VEL
LIN {X 0,Y 362.809,Z 187.683,A -85,B 0,C 180,E1 -13089.735,E2 -13089.735} C_VEL
LIN {X 0,Y 361.842,Z 182.415,A -85,B 0,C 180,E1 -13093.485,E2 -13093.485} C_VEL
LIN {X 0,Y 361.835,Z 182.412,A -85,B 0,C 180,E1 -13097.171,E2 -13097.171} C_VEL
LIN {X 0,Y 361.83,Z 182.412,A -85,B 0,C 180,E1 -13100.98,E2 -13100.98} C_VEL
LIN {X 0,Y 361.872,Z 182.408,A -85,B 0,C 180,E1 -13104.655,E2 -13104.655} C_VEL
LIN {X 0,Y 361.836,Z 182.414,A -85,B 0,C 180,E1 -13108.37,E2 -13108.37} C_VEL
LIN {X 0,Y 361.906,Z 182.405,A -85,B 0,C 180,E1 -13112.221,E2 -13112.221} C_VEL
LIN {X 0,Y 361.924,Z 182.399,A -85,B 0,C 180,E1 -13114.71,E2 -13114.71} C_VEL
LIN {X 0,Y 361.859,Z 182.408,A -85,B 0,C 180,E1 -13118.345,E2 -13118.345} C_VEL
LIN {X 0,Y 361.965,Z 182.396,A -85,B 0,C 180,E1 -13122.061,E2 -13122.061} C_VEL
LIN {X 0,Y 361.996,Z 182.391,A -85,B 0,C 180,E1 -13126.101,E2 -13126.101} C_VEL
LIN {X 0,Y 361.997,Z 182.391,A -85,B 0,C 180,E1 -13129.937,E2 -13129.937} C_VEL
LIN {X 0,Y 362.12,Z 182.379,A -85,B 0,C 180,E1 -13133.313,E2 -13133.313} C_VEL
LIN {X 0,Y 362.277,Z 182.355,A -85,B 0,C 180,E1 -13137.776,E2 -13137.776} C_VEL
LIN {X 0,Y 362.426,Z 182.337,A -85,B 0,C 180,E1 -13140,E2 -13140} C_VEL
LIN {X 0,Y 362.277,Z 182.356,A -85,B 0,C 180,E1 -13142.224,E2 -13142.224} C_VEL
LIN {X 0,Y 362.12,Z 182.379,A -85,B 0,C 180,E1 -13146.687,E2 -13146.687} C_VEL
LIN {X 0,Y 361.997,Z 182.392,A -85,B 0,C 180,E1 -13150.063,E2 -13150.063} C_VEL
LIN {X 0,Y 361.996,Z 182.393,A -85,B 0,C 180,E1 -13153.899,E2 -13153.899} C_VEL
LIN {X 0,Y 361.965,Z 182.398,A -85,B 0,C 180,E1 -13157.939,E2 -13157.939} C_VEL
LIN {X 0,Y 361.89,Z 182.406,A -85,B 0,C 180,E1 -13161.653,E2 -13161.653} C_VEL
LIN {X 0,Y 361.926,Z 182.4,A -85,B 0,C 180,E1 -13165.29,E2 -13165.29} C_VEL
LIN {X 0,Y 361.907,Z 182.406,A -85,B 0,C 180,E1 -13167.779,E2 -13167.779} C_VEL
LIN {X 0,Y 361.836,Z 182.415,A -85,B 0,C 180,E1 -13171.63,E2 -13171.63} C_VEL
LIN {X 0,Y 361.872,Z 182.411,A -85,B 0,C 180,E1 -13175.345,E2 -13175.345} C_VEL
LIN {X 0,Y 361.831,Z 182.415,A -85,B 0,C 180,E1 -13179.02,E2 -13179.02} C_VEL
LIN {X 0,Y 361.835,Z 182.414,A -85,B 0,C 180,E1 -13182.829,E2 -13182.829} C_VEL
LIN {X 0,Y 361.817,Z 182.412,A -85,B 0,C 180,E1 -13185.947,E2 -13185.947} C_VEL
LIN {X 0,Y 361.835,Z 182.412,A -85,B 0,C 180,E1 -13189.245,E2 -13189.245} C_VEL
LIN {X 0,Y 361.856,Z 182.408,A -85,B 0,C 180,E1 -13191.574,E2 -13191.574} C_VEL
LIN {X 0,Y 361.811,Z 182.42,A -85,B 0,C 180,E1 -13192.976,E2 -13192.976} C_VEL
LIN {X 0,Y 361.782,Z 185.1,A -85,B 0,C 180,E1 -13195.712,E2 -13195.712} C_VEL
LIN {X 0,Y 361.659,Z 188.474,A -85,B 0,C 180,E1 -13198.764,E2 -13198.764} C_VEL
LIN {X 0,Y 361.43,Z 192.422,A -85,B 0,C 180,E1 -13202.181,E2 -13202.181} C_VEL
LIN {X 0,Y 361.2,Z 197.177,A -85,B 0,C 180,E1 -13206.135,E2 -13206.135} C_VEL
LIN {X 0,Y 360.991,Z 202.151,A -85,B 0,C 180,E1 -13209.997,E2 -13209.997} C_VEL
LIN {X 0,Y 364.353,Z 215.488,A -85,B 0,C 180,E1 -13210.698,E2 -13210.698} C_VEL
LIN {X 0,Y 366.877,Z 227.423,A -85,B 0,C 180,E1 -13211.509,E2 -13211.509} C_VEL
LIN {X 0,Y 367.546,Z 232.963,A -85,B 0,C 180,E1 -13211.931,E2 -13211.931} C_VEL
LIN {X 0,Y 366.594,Z 244.487,A -85,B 0,C 180,E1 -13212.858,E2 -13212.858} C_VEL
LIN {X 0,Y 365.57,Z 255.475,A -85,B 0,C 180,E1 -13213.996,E2 -13213.996} C_VEL
LIN {X 0,Y 364.762,Z 264.868,A -85,B 0,C 180,E1 -13215.209,E2 -13215.209} C_VEL
LIN {X 0,Y 363.712,Z 273.708,A -85,B 0,C 180,E1 -13216.593,E2 -13216.593} C_VEL
LIN {X 0,Y 362.738,Z 282.327,A -85,B 0,C 180,E1 -13218.262,E2 -13218.262} C_VEL
LIN {X 0,Y 361.924,Z 289.198,A -85,B 0,C 180,E1 -13219.935,E2 -13219.935} C_VEL
LIN {X 0,Y 361.314,Z 294.697,A -85,B 0,C 180,E1 -13221.612,E2 -13221.612} C_VEL
LIN {X 0,Y 360.865,Z 299.858,A -85,B 0,C 180,E1 -13223.676,E2 -13223.676} C_VEL
LIN {X 0,Y 360.574,Z 303.152,A -85,B 0,C 180,E1 -13225.529,E2 -13225.529} C_VEL
LIN {X 0,Y 360.442,Z 304.55,A -85,B 0,C 180,E1 -13226.647,E2 -13226.647} C_VEL
LIN {X 0,Y 360.369,Z 306.155,A -85,B 0,C 180,E1 -13228.883,E2 -13228.883} C_VEL
LIN {X 0,Y 360.363,Z 306.387,A -85,B 0,C 180,E1 -13230,E2 -13230} C_VEL
LIN {X 0,Y 360.369,Z 306.198,A -85,B 0,C 180,E1 -13231.118,E2 -13231.118} C_VEL
LIN {X 0,Y 360.44,Z 304.648,A -85,B 0,C 180,E1 -13233.354,E2 -13233.354} C_VEL
LIN {X 0,Y 360.571,Z 303.291,A -85,B 0,C 180,E1 -13234.472,E2 -13234.472} C_VEL
LIN {X 0,Y 360.86,Z 300.097,A -85,B 0,C 180,E1 -13236.316,E2 -13236.316} C_VEL
LIN {X 0,Y 361.31,Z 294.985,A -85,B 0,C 180,E1 -13238.389,E2 -13238.389} C_VEL
LIN {X 0,Y 362.048,Z 288.55,A -85,B 0,C 180,E1 -13240.344,E2 -13240.344} C_VEL
LIN {X 0,Y 362.856,Z 281.478,A -85,B 0,C 180,E1 -13242.018,E2 -13242.018} C_VEL
LIN {X 0,Y 363.851,Z 272.665,A -85,B 0,C 180,E1 -13243.687,E2 -13243.687} C_VEL
LIN {X 0,Y 364.919,Z 263.617,A -85,B 0,C 180,E1 -13245.07,E2 -13245.07} C_VEL
LIN {X 0,Y 365.788,Z 253.82,A -85,B 0,C 180,E1 -13246.295,E2 -13246.295} C_VEL
LIN {X 0,Y 366.853,Z 242.454,A -85,B 0,C 180,E1 -13247.418,E2 -13247.418} C_VEL
LIN {X 0,Y 367.631,Z 232.629,A -85,B 0,C 180,E1 -13248.191,E2 -13248.191} C_VEL
LIN {X 0,Y 365.708,Z 221.393,A -85,B 0,C 180,E1 -13249.025,E2 -13249.025} C_VEL
LIN {X 0,Y 362.712,Z 208.631,A -85,B 0,C 180,E1 -13249.793,E2 -13249.793} C_VEL
LIN {X 0,Y 360.966,Z 202.024,A -85,B 0,C 180,E1 -13250.141,E2 -13250.141} C_VEL
LIN {X 0,Y 361.182,Z 197.328,A -85,B 0,C 180,E1 -13253.858,E2 -13253.858} C_VEL
LIN {X 0,Y 361.429,Z 192.564,A -85,B 0,C 180,E1 -13257.819,E2 -13257.819} C_VEL
LIN {X 0,Y 361.662,Z 188.602,A -85,B 0,C 180,E1 -13261.236,E2 -13261.236} C_VEL
LIN {X 0,Y 361.754,Z 186.693,A -85,B 0,C 180,E1 -13262.947,E2 -13262.947} C_VEL
LIN {X 0,Y 361.174,Z 185.764,A -85,B 0,C 180,E1 -13263.865,E2 -13263.865} C_VEL
LIN {X 0,Y 358.34,Z 184.524,A -85,B 0,C 180,E1 -13265.365,E2 -13265.365} C_VEL
LIN {X 0,Y 355.894,Z 183.683,A -85,B 0,C 180,E1 -13266.584,E2 -13266.584} C_VEL
LIN {X 0,Y 354.852,Z 183.323,A -85,B 0,C 180,E1 -13267.53,E2 -13267.53} C_VEL
LIN {X 0,Y 354.774,Z 183.292,A -85,B 0,C 180,E1 -13267.851,E2 -13267.851} C_VEL
LIN {X 0,Y 354.772,Z 183.295,A -85,B 0,C 180,E1 -13271.168,E2 -13271.168} C_VEL
LIN {X 0,Y 354.764,Z 183.292,A -85,B 0,C 180,E1 -13274.506,E2 -13274.506} C_VEL
LIN {X 0,Y 354.795,Z 183.288,A -85,B 0,C 180,E1 -13277.663,E2 -13277.663} C_VEL
LIN {X 0,Y 354.786,Z 183.292,A -85,B 0,C 180,E1 -13280.662,E2 -13280.662} C_VEL
LIN {X 0,Y 354.822,Z 183.286,A -85,B 0,C 180,E1 -13284.301,E2 -13284.301} C_VEL
LIN {X 0,Y 354.788,Z 183.288,A -85,B 0,C 180,E1 -13287.666,E2 -13287.666} C_VEL
LIN {X 0,Y 354.848,Z 183.281,A -85,B 0,C 180,E1 -13291.619,E2 -13291.619} C_VEL
LIN {X 0,Y 354.9,Z 183.279,A -85,B 0,C 180,E1 -13294.173,E2 -13294.173} C_VEL
LIN {X 0,Y 354.836,Z 183.285,A -85,B 0,C 180,E1 -13297.894,E2 -13297.894} C_VEL
LIN {X 0,Y 354.924,Z 183.276,A -85,B 0,C 180,E1 -13301.891,E2 -13301.891} C_VEL
LIN {X 0,Y 354.944,Z 183.273,A -85,B 0,C 180,E1 -13305.981,E2 -13305.981} C_VEL
LIN {X 0,Y 354.956,Z 183.272,A -85,B 0,C 180,E1 -13309.735,E2 -13309.735} C_VEL
LIN {X 0,Y 355.089,Z 183.253,A -85,B 0,C 180,E1 -13313.18,E2 -13313.18} C_VEL
LIN {X 0,Y 355.242,Z 183.233,A -85,B 0,C 180,E1 -13317.732,E2 -13317.732} C_VEL
LIN {X 0,Y 355.399,Z 183.212,A -85,B 0,C 180,E1 -13320,E2 -13320} C_VEL
LIN {X 0,Y 355.243,Z 183.231,A -85,B 0,C 180,E1 -13322.268,E2 -13322.268} C_VEL
LIN {X 0,Y 355.089,Z 183.256,A -85,B 0,C 180,E1 -13326.82,E2 -13326.82} C_VEL
LIN {X 0,Y 354.979,Z 183.266,A -85,B 0,C 180,E1 -13330.264,E2 -13330.264} C_VEL
LIN {X 0,Y 354.944,Z 183.27,A -85,B 0,C 180,E1 -13334.019,E2 -13334.019} C_VEL
LIN {X 0,Y 354.924,Z 183.274,A -85,B 0,C 180,E1 -13338.108,E2 -13338.108} C_VEL
LIN {X 0,Y 354.817,Z 183.289,A -85,B 0,C 180,E1 -13342.107,E2 -13342.107} C_VEL
LIN {X 0,Y 354.899,Z 183.278,A -85,B 0,C 180,E1 -13345.827,E2 -13345.827} C_VEL
LIN {X 0,Y 354.819,Z 183.288,A -85,B 0,C 180,E1 -13349.682,E2 -13349.682} C_VEL
LIN {X 0,Y 354.807,Z 183.292,A -85,B 0,C 180,E1 -13353.702,E2 -13353.702} C_VEL
LIN {X 0,Y 354.796,Z 183.288,A -85,B 0,C 180,E1 -13356.46,E2 -13356.46} C_VEL
LIN {X 0,Y 354.799,Z 183.292,A -85,B 0,C 180,E1 -13359.419,E2 -13359.419} C_VEL
LIN {X 0,Y 354.789,Z 183.29,A -85,B 0,C 180,E1 -13362.867,E2 -13362.867} C_VEL
LIN {X 0,Y 354.844,Z 183.45,A -85,B 0,C 180,E1 -13366.284,E2 -13366.284} C_VEL
LIN {X 0,Y 355.576,Z 187.58,A -85,B 0,C 180,E1 -13369.288,E2 -13369.288} C_VEL
LIN {X 0,Y 356.232,Z 191.958,A -85,B 0,C 180,E1 -13372.295,E2 -13372.295} C_VEL
LIN {X 0,Y 356.351,Z 196.351,A -85,B 0,C 180,E1 -13375.114,E2 -13375.114} C_VEL
LIN {X 0,Y 355.901,Z 201.302,A -85,B 0,C 180,E1 -13378.117,E2 -13378.117} C_VEL
LIN {X 0,Y 355.286,Z 207.328,A -85,B 0,C 180,E1 -13381.657,E2 -13381.657} C_VEL
LIN {X 0,Y 354.718,Z 213.85,A -85,B 0,C 180,E1 -13385.413,E2 -13385.413} C_VEL
LIN {X 0,Y 354.236,Z 220.824,A -85,B 0,C 180,E1 -13389.381,E2 -13389.381} C_VEL
LIN {X 0,Y 354.221,Z 221.024,A -85,B 0,C 180,E1 -13389.494,E2 -13389.494} C_VEL
LIN {X 0,Y 357.148,Z 235.473,A -85,B 0,C 180,E1 -13390.215,E2 -13390.215} C_VEL
LIN {X 0,Y 359.11,Z 248.524,A -85,B 0,C 180,E1 -13391.068,E2 -13391.068} C_VEL
LIN {X 0,Y 360.001,Z 257.67,A -85,B 0,C 180,E1 -13391.799,E2 -13391.799} C_VEL
LIN {X 0,Y 358.799,Z 270.111,A -85,B 0,C 180,E1 -13392.913,E2 -13392.913} C_VEL
LIN {X 0,Y 357.73,Z 279.942,A -85,B 0,C 180,E1 -13394.035,E2 -13394.035} C_VEL
LIN {X 0,Y 356.684,Z 289.913,A -85,B 0,C 180,E1 -13395.45,E2 -13395.45} C_VEL
LIN {X 0,Y 355.617,Z 299.582,A -85,B 0,C 180,E1 -13397.154,E2 -13397.154} C_VEL
LIN {X 0,Y 354.7,Z 307.279,A -85,B 0,C 180,E1 -13398.861,E2 -13398.861} C_VEL
LIN {X 0,Y 353.991,Z 314.38,A -85,B 0,C 180,E1 -13400.861,E2 -13400.861} C_VEL
LIN {X 0,Y 353.557,Z 319.105,A -85,B 0,C 180,E1 -13402.576,E2 -13402.576} C_VEL
LIN {X 0,Y 353.33,Z 322.718,A -85,B 0,C 180,E1 -13404.292,E2 -13404.292} C_VEL
LIN {X 0,Y 353.299,Z 324.584,A -85,B 0,C 180,E1 -13405.436,E2 -13405.436} C_VEL
